	csp_main.i_csp_data_ref^.Production.GoodCasesNoReset	:=	UDINT_TO_DINT(csp_case_main_statistics.logsect.hmi_unresettable_sampled_counters.total_good_products);
	
	csp_main.i_csp_data_ref^.Production.GoodUnitsNoReset	:=	UDINT_TO_DINT(csp_case_main_statistics.logsect.hmi_unresettable_sampled_counters.total_good_products)
																*
																csp_main_brand.case_pattern.case_pattern_L
																*
																csp_main_brand.case_pattern.case_pattern_W;
																
	csp_main.i_csp_data_ref^.Production.TotalUnits			:=	(csp_customerInterfaces.CasePacker.Production.GoodUnits + csp_customerInterfaces.CasePacker.Production.TotalScrapUnits); //Cartoni Ricevuti a monte del metering belt per un ordine, a prescindere che andranno scartati o meno dal pusher
	
	csp_main.i_csp_data_ref^.Production.TotalUnitsNoReset	:=	(
																UDINT_TO_DINT(csp_case_main_statistics.logsect.hmi_unresettable_sampled_counters.total_good_products)
																+
																UDINT_TO_DINT(csp_case_main_statistics.logsect.hmi_unresettable_sampled_counters.total_rejected)
																)
																	*
																	csp_main_brand.case_pattern.case_pattern_L
																	*
																	csp_main_brand.case_pattern.case_pattern_W; //Cartoni Ricevuti a monte del metering belt, a prescindere che andranno scartati o meno dal pusher
																
	csp_main.i_csp_data_ref^.Production.TotalScrapUnits		:=	UDINT_TO_DINT(csp_case_main_statistics.logsect.hmi_shift_independent_sampled_counters.total_rejected)
																*
																csp_main_brand.case_pattern.case_pattern_L
																*
																csp_main_brand.case_pattern.case_pattern_W;
																
	csp_main.i_csp_data_ref^.Production.TotalOrderTime		:= 	UDINT_TO_DINT(mes_elapsed_time_1_npr / 60); 	
	csp_main.i_csp_data_ref^.Production.TotalRunningTime 	:=	UDINT_TO_DINT(mes_elapsed_time_2_npr / 60); 
	
	//Divide by zero protections
	IF UDINT_TO_DINT(csp_case_main_statistics.logsect.hmi_shift_independent_sampled_counters.total_good_products) <> 0
	THEN
	csp_main.i_csp_data_ref^.Production.PercentScrapUnits	:=	(		//Rejected Cases
																		UDINT_TO_DINT(csp_case_main_statistics.logsect.hmi_shift_independent_sampled_counters.total_rejected)
																		/ 
																		UDINT_TO_DINT(csp_case_main_statistics.logsect.hmi_shift_independent_sampled_counters.total_good_products)
																)		//Good Cases
																*
																100;
	END_IF																
	
	csp_main.i_csp_data_ref^.Production.Rejects.Infeed_waterfall	:=	//Barcode Rejects
																		UDINT_TO_DINT(csp_case_main_statistics.logsect.hmi_shift_independent_sampled_counters.auxiliary_counters[1])
																		+
																		//High Load Rejects
																		UDINT_TO_DINT(csp_case_main_statistics.logsect.hmi_shift_independent_sampled_counters.auxiliary_counters[2]);
																			
	csp_main.i_csp_data_ref^.Production.Rejects.Accumulator	:=		//Crosspush Low-load
																		UDINT_TO_DINT(csp_case_main_statistics.logsect.hmi_shift_independent_sampled_counters.auxiliary_counters[3])
																		+
																	//Crosspush High-load
																		UDINT_TO_DINT(csp_case_main_statistics.logsect.hmi_shift_independent_sampled_counters.auxiliary_counters[4]);												
																			
	csp_main.i_csp_data_ref^.Production.Rejects.Case_Feed	:=		//Case Feed Reject
																		UDINT_TO_DINT(csp_case_main_statistics.logsect.hmi_shift_independent_sampled_counters.auxiliary_counters[5]);

	csp_main.i_csp_data_ref^.Production.Rejects.Discharge	:=		//Rejected cases at discharge
																		UDINT_TO_DINT(csp_case_main_statistics.logsect.hmi_shift_independent_sampled_counters.total_rejected);
	
	csp_main.i_csp_data_ref^.Production.Rejects.TBD5		:=		TEST_DINT;
	csp_main.i_csp_data_ref^.Production.Rejects.Sample		:=		TEST_DINT;
	
	(*from RAJones MIX - MARCO *)
	
	csp_main.i_csp_data_ref^.Start.PeakWait 				:= 	FALSE;
	csp_main.i_csp_data_ref^.Start.Ramp 					:= 	FALSE;	
	csp_main.i_csp_data_ref^.Start.Request 					:= 	FALSE;	
	
	csp_main.i_csp_data_ref^.Status.NextJob 				:= 	TEST_DINT;;
	csp_main.i_csp_data_ref^.Status.Running 				:= 	motorization_manager_is_execute(csp_main_motorization_manager.motm);

	csp_main.i_csp_data_ref^.Status.Blocked.Downstream 		:= 	message_is_on(csp_case_discharge_reject_sensors.downstream_backup_hold_aem);
	csp_main.i_csp_data_ref^.Status.Blocked.Reject 			:= 	message_is_on(csp_case_discharge_reject_sensors.consecutive_blocked_reject_aem);
	csp_main.i_csp_data_ref^.Status.Blocked.Waste 			:= 	message_is_on(csp_transfer_crosspusher_reject.backup_di_dchk.alarm_asm.message)
																OR
																message_is_on(csp_transfer_infeed_reject.bin_full_dchk.alarm_asm.message);

	csp_main.i_csp_data_ref^.Status.Faulted.CaseBlanks		:= 	csp_case_feed_magazine.AML_Faulted;;
	
	csp_main.i_csp_data_ref^.Status.Faulted.Main 			:= 	machine_is_stopped(csp.mch)
																AND 
																csp_main_interface.alarm_id <> 430 // SERVICE CYCLE STOP FOR CASE SIDE
																AND 
																csp_main_interface.alarm_id <> 431 // CYCLE STOP FOR CASE SIDE	
																AND 
																csp_main_interface.alarm_id <> 768 // SERVICE CYCLE STOP FOR TRANSFER SIDE
																AND 
																csp_main_interface.alarm_id <> 769;// CYCLE STOP FOR TRANSFER SIDE	

	csp_main.i_csp_data_ref^.Status.Rate.Actual				:= 	LREAL_TO_INT(csp_main_motorization_manager.motm.actual_velocity);
	
	csp_main.i_csp_data_ref^.Status.Rate.Target				:= 	LREAL_TO_INT(csp_main_motorization_manager.motm.actual_velocity_setpoint);
	
	csp_main.i_csp_data_ref^.Status.Starved.CaseBlanks 		:= 	message_is_on(csp_case_feed_magazine_level_zonemin.magazine_level_zone_min_wem); //MARCO: PE presente nella presa cases
	csp_main.i_csp_data_ref^.Status.Starved.Glue 			:= 	NOT digital_input_is_active(csp_case_glue_hotmelt.level_ok_di);
	csp_main.i_csp_data_ref^.Status.Starved.Labels 			:= 	TEST_BOOL; //MARCO: inserire out_of_label che possiamo leggere dallo step 4 della cartoner
	csp_main.i_csp_data_ref^.Status.Starved.Units 			:= 	csp_transfer_infeed_clamp.min_prime; //MARCO: indica che il livello dei cartoni è inferiore al min, oltre ad altri check da verificare se siano corretti (RAJones)
	
	csp_main.i_csp_data_ref^.Status.Stop.AutoReason 		:= 	csp_main_interface.alarm_id; 
	csp_main.i_csp_data_ref^.Status.Stop.Estop 				:= 	//machine_is_stop_emergency_active(csp.mch);
																NOT safety_integrated_series_is_safely_closed(csp_case_main_safety_emergency.sis)
																OR
																NOT safety_integrated_series_is_safely_closed(csp_transfer_main_safety_emergency.sis);
																
	csp_main.i_csp_data_ref^.Status.Stop.Guard 				:= 	NOT safety_integrated_series_is_safely_closed(csp_case_main_safety_guards.sis) OR NOT safety_integrated_series_is_safely_closed(csp_transfer_main_safety_guards.sis);
	csp_main.i_csp_data_ref^.Status.Stop.Operator 			:= 	message_is_on(csp_case_main_services_pushbuttons.stop_dchk.alarm_asm.message)
																OR
																message_is_on(csp_case_main_services_pushbuttons.service_stop_dchk.alarm_asm.message)
																OR
																message_is_on(csp_transfer_main_services_pushbuttons.stop_dchk.alarm_asm.message)
																OR
																message_is_on(csp_transfer_main_services_pushbuttons.service_stop_dchk.alarm_asm.message);
	
	csp_main.i_csp_data_ref^.Status.RunOut 					:= 	csp_main_motorization.empty_command;
	csp_main.i_csp_data_ref^.Status.RunOutComplete 			:=	message_is_on(csp_case_virtualMaster.runout_complete)
																AND csp_case_main_services.end_production
																OR
																p_last_case;
	
ELSE
	mes_elapsed_time_1_npr	:= 0;
	mes_elapsed_time_2_npr	:= 0;
END_IF
END_ACTION

END_PROGRAM

// ---- Application/CSP/Main/Phase Manager/csp_main_phaseManager_run_out.TcPOU
(*********************************** G.D S.p.A. - Technical Department ***********************************
============= PROGRAM INFO ============
FOLDER:             TBD
MACHINES INVOLVED:  TBD 

============= DESCRIPTION =============
WN phase manager program

============= REVISIONS ===============
Date		Version	 	Author      	Description             
----------	-------		------------  	--------------------------------------------
2021/03/18 	0000.01	 	S.Uccellari 	Creation of the PRG
**********************************************************************************************************)
(*$R
	process_ref := prc;
$*)
PROGRAM csp_main_phaseManager_run_out
VAR
	prc:												process;
	prc_path:											STRING;
	
	fsm_enable_conditions:								BOOL;
	fsm_status:											INT;
	
	rejects_for_low_weight_init_cnt:					UDINT;
	rejects_for_low_weight_cnt:							UDINT;	
	rejects_for_low_weight_limit_npr:					UDINT;		(*$P desc := run out - cups under weight; $*)

	confirm_run_out_mode_dpr:							BOOL;		(*$P $*)	
	confirm_run_out_mode_pow:							parameter_overwrite;	
	confirm_run_out_mode_visibility:					INT := 1; 	(*$H_R	desc := visibility; $*)

	low_weight_limit_asm:								message;	
	run_out_complete_asm:								message;	
	
	
	run_out_running:									BOOL;
	run_out_done:										BOOL;
	
END_VAR

_read_var_input();

_object_manager();

IF NOT objects_running()
THEN
	RETURN;	
END_IF

_read_process_image();

_mode_manager();

CASE process_get_mode(prc) of
	MODE_ABSENT,
	MODE_INACTIVE:
		RETURN;
	MODE_TEST:
		_handle_process_test();
END_CASE

_set_runtime_properties();

(********************************* BODY *********************************)

(************************************************************************)

(**************************** PROGRAM HANDLER ***************************)
run_cycle();
(************************************************************************)

_handle_messages();

_write_output();

ACTION _handle_messages:
;
END_ACTION

ACTION _handle_process_test:
;
END_ACTION

ACTION _mode_manager:
IF process_mode_req_is_pending(prc)
THEN
    process_apply_mode_req_first_step(prc);
    CASE process_get_mode(prc) OF
        MODE_TO_ABSENT:
			;
        MODE_TO_INACTIVE:
			;
        MODE_TO_TEST:
			;
        MODE_TO_OPERATIONAL:
			;
    END_CASE
    process_apply_mode_req_second_step(prc);
END_IF
END_ACTION

ACTION _object_manager:
IF objects_initialization()
THEN
	sub_process_init(
		object_name					:= 'csp_main_phaseManager_run_out.prc', 
		process						:= csp_main_phaseManager.prc, 
		CONVERSION_this				:= prc);
		
	prc_path 						:= process_get_path(prc);
	
	parameter_overwrite_bool_init(
		object_name								:= CONCAT(prc_path, '_confirm_run_out_mode_pow'), 
		parameter								:= confirm_run_out_mode_dpr, 
		process									:= prc, 
		CONVERSION_this							:= confirm_run_out_mode_pow);		

	process_message_init(
		object_name					:= CONCAT(prc_path, '_low_weight_limit_asm'), 
		behaviour					:= MESSAGE_BEHAVIOUR_STATE, 
		reset_timeout				:= 0, 
		disableable					:= FALSE, 
		individual_reset			:= FALSE, 
		machine_reaction			:= MACHINE_REACTION_NORMAL_STOP, 
		typology					:= MESSAGE_TYPOLOGY_ABNORMAL, 
		process						:= prc, 
		CONVERSION_this				:= low_weight_limit_asm);

	process_message_init(
		object_name					:= CONCAT(prc_path, '_run_out_complete_asm'), 
		behaviour					:= MESSAGE_BEHAVIOUR_EVENT, 
		reset_timeout				:= 0, 
		disableable					:= FALSE, 
		individual_reset			:= FALSE, 
		machine_reaction			:= MACHINE_REACTION_NORMAL_STOP, 
		typology					:= MESSAGE_TYPOLOGY_ABNORMAL, 
		process						:= prc, 
		CONVERSION_this				:= run_out_complete_asm);


		

END_IF

IF objects_running()
THEN
	process_cycle(prc);
END_IF
END_ACTION

ACTION _read_process_image:
;
END_ACTION

ACTION _read_var_input:
;
END_ACTION

ACTION _set_runtime_properties:
;
END_ACTION

ACTION _write_output:
;
END_ACTION

ACTION run_cycle:
IF	csp_main_phaseManager.fsm_status = CSP_MAIN_PHASE_MANAGER_STATUS_UNDEFINED_0
	AND
	csp_main_phaseManager.p_mes_interface_enable
THEN	
	fsm_status := 0;
END_IF

fsm_enable_conditions :=
	(
		csp_main_phaseManager.fsm_status
		=
		CSP_MAIN_PHASE_MANAGER_STATUS_RUNOUT_60
	);
	
IF	NOT fsm_enable_conditions
THEN
	process_message_reset(low_weight_limit_asm);	
	IF	run_out_running	
	THEN
		fsm_status := 666;
	END_IF;	
END_IF

CASE fsm_status OF
	0:
		confirm_run_out_mode_visibility := 1;	
		csp_main.i_csp_data_ref^.Status.RunOutComplete := FALSE;
		IF fsm_enable_conditions
		THEN
			run_out_done := FALSE;
			run_out_running := TRUE;
			fsm_status := 20;
		END_IF
		
	20:		
		fsm_status := 30;			
		

	30:	
		fsm_status := 40;	

	40:
		confirm_run_out_mode_visibility := 1;
		csp_main.i_csp_data_ref^.Status.RunOut := TRUE; (* use this to empty the filler *)

			fsm_status := 555;


	50: 
		;
		(*IF filler_empty
		THEN
			process_message_set(
				errorID_1			:= 1, 
				errorID_2			:= 0, 
				errorID_3			:= 0, 
				CONVERSION_this		:= run_out_complete_asm);

			run_out step1 AND run out cartoner
			
			fsm_status := 555;
		END_IF*)
		
		
	555:
		csp_main.i_csp_data_ref^.Status.RunOut := FALSE;	
		csp_main.i_csp_data_ref^.Status.RunOutComplete := TRUE;
		run_out_running := FALSE;
		run_out_done := TRUE;
		confirm_run_out_mode_visibility := 1;
		
		IF	csp_main.i_filler_upstream_coffee //MARCO 0904
		THEN
			run_out_running := FALSE;
			run_out_done := FALSE;
			fsm_status := 0;
		END_IF		
		
	666:
		run_out_running := FALSE;
		run_out_done := FALSE;
		confirm_run_out_mode_visibility := 1;		
		csp_main.i_csp_data_ref^.Status.RunOut := FALSE;		
		csp_main.i_csp_data_ref^.Status.RunOutComplete := FALSE;
		//IF NOT csp_main.i_upstream_coffee^.Down //MARCO 0904
		//THEN
			fsm_status := 0;
		//END_IF
END_CASE
END_ACTION

END_PROGRAM

// ---- Application/CSP/Main/Phase Manager/Snapshot/csp_main_phaseManager_set_snapshot.TcPOU
(*********************************** G.D S.p.A. - Technical Department ***********************************
============= PROGRAM INFO ============
FOLDER:             TBD
MACHINES INVOLVED:  TBD 

============= DESCRIPTION =============
WU phase manager snapshot set function

============= REVISIONS ===============
Date		Version	 	Author      	Description             
----------	-------		------------  	--------------------------------------------
2020/06/19 	0000.00	 	G.Cera 			Creation of the PRG

**********************************************************************************************************)

FUNCTION csp_main_phaseManager_set_snapshot : VOID
VAR_INPUT
    errorID_1:				DINT;			(* Field for specify the faults code or enter
								   				more message info *)
    errorID_2:				DINT;			(* Field for specify the faults code or enter
								   				more message info *)
    errorID_3:				DINT;			(* Field for specify the faults code or enter
								   				more message info *)
	reason:					STRING := '';

	job_not_scheduled:		BOOL;
	
	job_pending:			BOOL;
	
END_VAR

VAR_IN_OUT
    CONVERSION_this:		csp_main_phaseManager_snapshot;
								(* csp_main_phaseManager_snapshot snapshot reference *)
END_VAR

IF	message_set(
		errorID_1		:= errorID_1, 
		errorID_2		:= errorID_2, 
		errorID_3		:= errorID_3, 
		CONVERSION_this	:= CONVERSION_this.message)
THEN
	CONVERSION_this.reason 				:= reason;
	CONVERSION_this.job_not_scheduled	:= job_not_scheduled;
	CONVERSION_this.job_pending			:= job_pending;
END_IF

END_FUNCTION

// ---- Application/CSP/Main/Phase Manager/Snapshot/csp_main_phaseManager_warning_set_snapshot.TcPOU
(*********************************** G.D S.p.A. - Technical Department ***********************************
============= PROGRAM INFO ============
FOLDER:             TBD
MACHINES INVOLVED:  TBD 

============= DESCRIPTION =============
WU phase manager snapshot set function

============= REVISIONS ===============
Date		Version	 	Author      	Description             
----------	-------		------------  	--------------------------------------------
2020/06/19 	0000.00	 	G.Cera 			Creation of the PRG

**********************************************************************************************************)

FUNCTION csp_main_phaseManager_warning_set_snapshot : VOID
VAR_INPUT
    errorID_1:				DINT;			(* Field for specify the faults code or enter
								   				more message info *)
    errorID_2:				DINT;			(* Field for specify the faults code or enter
								   				more message info *)
    errorID_3:				DINT;			(* Field for specify the faults code or enter
								   				more message info *)
	reason:					STRING := '';

	maintenance_job_active:	BOOL;
		
END_VAR

VAR_IN_OUT
    CONVERSION_this:		csp_main_phaseManager_warning_snapshot;
								(* csp_main_phaseManager_snapshot snapshot reference *)
END_VAR

IF	message_set(
		errorID_1		:= errorID_1, 
		errorID_2		:= errorID_2, 
		errorID_3		:= errorID_3, 
		CONVERSION_this	:= CONVERSION_this.message)
THEN
	CONVERSION_this.w_reason 					:= reason;
	CONVERSION_this.maintenance_job_active	:= maintenance_job_active;
END_IF

END_FUNCTION

// ---- Application/CSP/Main/Phase Manager/Snapshot/csp_main_phMan_start_job_set_snapshot.TcPOU
(*********************************** G.D S.p.A. - Technical Department ***********************************
============= PROGRAM INFO ============
FOLDER:             TBD
MACHINES INVOLVED:  TBD 

============= DESCRIPTION =============
WU phase manager snapshot set function

============= REVISIONS ===============
Date		Version	 	Author      	Description             
----------	-------		------------  	--------------------------------------------
2020/06/19 	0000.00	 	G.Cera 			Creation of the PRG

**********************************************************************************************************)

FUNCTION csp_main_phMan_start_job_set_snapshot : VOID
VAR_INPUT
    errorID_1:				DINT;			(* Field for specify the faults code or enter
								   				more message info *)
    errorID_2:				DINT;			(* Field for specify the faults code or enter
								   				more message info *)
    errorID_3:				DINT;			(* Field for specify the faults code or enter
								   				more message info *)
	reason:					STRING := '';

	order_valid:			BOOL;
	
	product_valid:			BOOL;
	
	recipe_valid:			BOOL;
	
	materials_valid:		BOOL;
	
	mark_valid:				BOOL;	
	
END_VAR

VAR_IN_OUT
    CONVERSION_this:		csp_main_phMan_start_job_snapshot;
								(* csp_main_phaseManager_snapshot snapshot reference *)
END_VAR

IF	message_set(
		errorID_1		:= errorID_1, 
		errorID_2		:= errorID_2, 
		errorID_3		:= errorID_3, 
		CONVERSION_this	:= CONVERSION_this.message)
THEN
	CONVERSION_this.sj_reason 				:= reason;
	CONVERSION_this.order_valid			:= order_valid;
	CONVERSION_this.recipe_valid		:= recipe_valid;
	CONVERSION_this.product_valid		:= product_valid;
	CONVERSION_this.materials_valid		:= materials_valid;
	CONVERSION_this.mark_valid			:= mark_valid;
END_IF

END_FUNCTION

// ---- Application/CSP/Main/Phase Manager/Snapshot/csp_main_phMan_start_job_init_snapshot.TcPOU
(*********************************** G.D S.p.A. - Technical Department ***********************************
============= PROGRAM INFO ============
FOLDER:             TBD
MACHINES INVOLVED:  TBD 

============= DESCRIPTION =============
WU phase manager snapshot init function

============= REVISIONS ===============
Date		Version	 	Author      	Description             
----------	-------		------------  	--------------------------------------------
2020/06/19 	0000.00	 	G.Cera 			Creation of the PRG

**********************************************************************************************************)

FUNCTION csp_main_phMan_start_job_init_snapshot : VOID
VAR_INPUT	
	message_name:			STRING(MAX_OBJ_NAME_LENGTH);
	behaviour:				message_behaviour_enum;			(* Message type. State or event *)
	reset_timeout:			UDINT;							(* Timeout of reset attempt valid for messages
															   with <a href="#message_behaviour_enum"><i>behaviour</i></a>
															   = MESSAGE_BEHAVIOUR_TRY_AND_CHECK *)
    disableable:        	BOOL;							(* Indicates the possibility
																to disable the message by HMI *)
    individual_reset:   	BOOL;							(* Need explicit reset by
																HMI for acknowlege the message.
																TRUE = individual_reset *)
    machine_reaction:		machine_reaction_enum;			(* Machine stop type.(emergency, normal,
																on phase, ...) *)
    typology:				message_typology_enum;			(* <a href="#message_typology_enum"><i>typology</i></a> *)	
END_VAR

VAR_IN_OUT
    process:                process;                    	(*$ <a href="#process_object"><i>process</i></a> membership $*)
	CONVERSION_this:		csp_main_phMan_start_job_snapshot;			
END_VAR

process_message_init(
	object_name 		:= message_name,
	behaviour 			:= behaviour,
	reset_timeout 		:= reset_timeout,
	disableable 		:= disableable,
	individual_reset 	:= individual_reset,
	machine_reaction 	:= machine_reaction,
	typology			:= typology,
	process 			:= process,
	CONVERSION_this 	:= CONVERSION_this.message);

CONVERSION_this.sj_reason := '';
CONVERSION_this.order_valid := FALSE;
CONVERSION_this.product_valid := FALSE;
CONVERSION_this.recipe_valid := FALSE;
CONVERSION_this.materials_valid := FALSE;
CONVERSION_this.mark_valid := FALSE;

END_FUNCTION

// ---- Application/CSP/Main/Phase Manager/Snapshot/csp_main_phaseManager_init_snapshot.TcPOU
(*********************************** G.D S.p.A. - Technical Department ***********************************
============= PROGRAM INFO ============
FOLDER:             TBD
MACHINES INVOLVED:  TBD 

============= DESCRIPTION =============
WU phase manager snapshot init function

============= REVISIONS ===============
Date		Version	 	Author      	Description             
----------	-------		------------  	--------------------------------------------
2020/06/19 	0000.00	 	G.Cera 			Creation of the PRG

**********************************************************************************************************)

FUNCTION csp_main_phaseManager_init_snapshot : VOID
VAR_INPUT	
	message_name:			STRING(MAX_OBJ_NAME_LENGTH);
	behaviour:				message_behaviour_enum;			(* Message type. State or event *)
	reset_timeout:			UDINT;							(* Timeout of reset attempt valid for messages
															   with <a href="#message_behaviour_enum"><i>behaviour</i></a>
															   = MESSAGE_BEHAVIOUR_TRY_AND_CHECK *)
    disableable:        	BOOL;							(* Indicates the possibility
																to disable the message by HMI *)
    individual_reset:   	BOOL;							(* Need explicit reset by
																HMI for acknowlege the message.
																TRUE = individual_reset *)
    machine_reaction:		machine_reaction_enum;			(* Machine stop type.(emergency, normal,
																on phase, ...) *)
    typology:				message_typology_enum;			(* <a href="#message_typology_enum"><i>typology</i></a> *)	
END_VAR

VAR_IN_OUT
    process:                process;                    	(*$ <a href="#process_object"><i>process</i></a> membership $*)
	CONVERSION_this:		csp_main_phaseManager_snapshot;			
END_VAR

process_message_init(
	object_name 		:= message_name,
	behaviour 			:= behaviour,
	reset_timeout 		:= reset_timeout,
	disableable 		:= disableable,
	individual_reset 	:= individual_reset,
	machine_reaction 	:= machine_reaction,
	typology			:= typology,
	process 			:= process,
	CONVERSION_this 	:= CONVERSION_this.message);

CONVERSION_this.reason := '';
CONVERSION_this.job_not_scheduled := FALSE;
CONVERSION_this.job_pending := FALSE;

END_FUNCTION

// ---- Application/CSP/Main/Phase Manager/Snapshot/csp_main_phaseManager_warning_init_snapshot.TcPOU
(*********************************** G.D S.p.A. - Technical Department ***********************************
============= PROGRAM INFO ============
FOLDER:             TBD
MACHINES INVOLVED:  TBD 

============= DESCRIPTION =============
WU phase manager snapshot init function

============= REVISIONS ===============
Date		Version	 	Author      	Description             
----------	-------		------------  	--------------------------------------------
2020/06/19 	0000.00	 	G.Cera 			Creation of the PRG

**********************************************************************************************************)

FUNCTION csp_main_phaseManager_warning_init_snapshot : VOID
VAR_INPUT	
	message_name:			STRING(MAX_OBJ_NAME_LENGTH);
	behaviour:				message_behaviour_enum;			(* Message type. State or event *)
	reset_timeout:			UDINT;							(* Timeout of reset attempt valid for messages
															   with <a href="#message_behaviour_enum"><i>behaviour</i></a>
															   = MESSAGE_BEHAVIOUR_TRY_AND_CHECK *)
    disableable:        	BOOL;							(* Indicates the possibility
																to disable the message by HMI *)
    individual_reset:   	BOOL;							(* Need explicit reset by
																HMI for acknowlege the message.
																TRUE = individual_reset *)
    machine_reaction:		machine_reaction_enum;			(* Machine stop type.(emergency, normal,
																on phase, ...) *)
    typology:				message_typology_enum;			(* <a href="#message_typology_enum"><i>typology</i></a> *)	
END_VAR

VAR_IN_OUT
    process:                process;                    	(*$ <a href="#process_object"><i>process</i></a> membership $*)
	CONVERSION_this:		csp_main_phaseManager_warning_snapshot;			
END_VAR

process_message_init(
	object_name 		:= message_name,
	behaviour 			:= behaviour,
	reset_timeout 		:= reset_timeout,
	disableable 		:= disableable,
	individual_reset 	:= individual_reset,
	machine_reaction 	:= machine_reaction,
	typology			:= typology,
	process 			:= process,
	CONVERSION_this 	:= CONVERSION_this.message);

CONVERSION_this.w_reason := '';
CONVERSION_this.maintenance_job_active := FALSE;

END_FUNCTION

// ---- Application/CSP/Main/Phase Manager/csp_main_phaseManager_end_job.TcPOU
(*********************************** G.D S.p.A. - Technical Department ***********************************
============= PROGRAM INFO ============
FOLDER:             TBD
MACHINES INVOLVED:  TBD 

============= DESCRIPTION =============
WN phase manager program

============= REVISIONS ===============
Date		Version	 	Author      	Description             
----------	-------		------------  	--------------------------------------------
2021/03/18 	0000.01	 	S.Uccellari 	Creation of the PRG
**********************************************************************************************************)
(*$R
	process_ref := prc;
$*)
PROGRAM csp_main_phaseManager_end_job
VAR
	prc:												process;
	prc_path:											STRING;
	
	fsm_enable_conditions:								BOOL;
	fsm_status:											INT;
	
	cycle_disable_from_mes_asm:							message;	
	
	end_job_running:									BOOL;
	end_job_done:										BOOL;
	
	i_start_job_done:									POINTER TO BOOL;	
	i_run_out_done:										POINTER TO BOOL;	
	
	debug_mes_endJobReq:								BOOL;		
	
END_VAR

_read_var_input();

_object_manager();

IF NOT objects_running()
THEN
	RETURN;	
END_IF

_read_process_image();

_mode_manager();

CASE process_get_mode(prc) of
	MODE_ABSENT,
	MODE_INACTIVE:
		RETURN;
	MODE_TEST:
		_handle_process_test();
END_CASE

_set_runtime_properties();

(********************************* BODY *********************************)

(************************************************************************)

(**************************** PROGRAM HANDLER ***************************)
run_cycle();
(************************************************************************)

_handle_messages();

_write_output();

ACTION _handle_messages:
;
END_ACTION

ACTION _handle_process_test:
;
END_ACTION

ACTION _mode_manager:
IF process_mode_req_is_pending(prc)
THEN
    process_apply_mode_req_first_step(prc);
    CASE process_get_mode(prc) OF
        MODE_TO_ABSENT:
			;
        MODE_TO_INACTIVE:
			;
        MODE_TO_TEST:
			;
        MODE_TO_OPERATIONAL:
			;
    END_CASE
    process_apply_mode_req_second_step(prc);
END_IF
END_ACTION

ACTION _object_manager:
IF objects_initialization()
THEN
	sub_process_init(
		object_name					:= 'csp_main_phaseManager_end_job.prc', 
		process						:= csp_main_phaseManager.prc, 
		CONVERSION_this				:= prc);
		
	prc_path 						:= process_get_path(prc);
	
	process_message_init(
		object_name					:= CONCAT(prc_path, '_cycle_disable_from_mes_asm'), 
		behaviour					:= MESSAGE_BEHAVIOUR_EVENT, 
		reset_timeout				:= 0, 
		disableable					:= FALSE, 
		individual_reset			:= FALSE, 
		machine_reaction			:= MACHINE_REACTION_NORMAL_STOP, 
		typology					:= MESSAGE_TYPOLOGY_ABNORMAL, 
		process						:= prc, 
		CONVERSION_this				:= cycle_disable_from_mes_asm);



END_IF

IF objects_running()
THEN
	process_cycle(prc);
END_IF
END_ACTION

ACTION _read_process_image:
;
END_ACTION

ACTION _read_var_input:
i_start_job_done 	:= ADR(csp_main_phaseManager_startJob.start_job_done);
i_run_out_done		:= ADR(csp_main_phaseManager_run_out.run_out_done);
END_ACTION

ACTION _set_runtime_properties:
;
END_ACTION

ACTION _write_output:
;
END_ACTION

ACTION run_cycle:
IF	csp_main_phaseManager.fsm_status = CSP_MAIN_PHASE_MANAGER_STATUS_UNDEFINED_0
THEN	
	fsm_status := 0;
END_IF

fsm_enable_conditions :=
	(
		csp_main_phaseManager.fsm_status
		=
		CSP_MAIN_PHASE_MANAGER_STATUS_END_JOB_70
	);
	
IF	NOT fsm_enable_conditions
THEN
	IF	end_job_running	
	THEN
		fsm_status := 666;
	END_IF;	
END_IF

CASE fsm_status OF
	0:	
		IF	fsm_enable_conditions
		THEN
				process_message_set(
					errorID_1			:= 1, 
					errorID_2			:= 0, 
				errorID_3			:= 0, 
					CONVERSION_this		:= cycle_disable_from_mes_asm);		
			
				end_job_done := FALSE;
				end_job_running := TRUE;
				fsm_status := 10;	
		END_IF	
		
	
	10:
		IF	csp_main.i_end_job_request
		THEN	
			log_section_upd_and_reset_factory_driven(csp_case_main_statistics.logsect);				
			csp_main.i_csp_data_ref^.Status.Job := 1;
			csp_main.i_cartons_count := 0;
			csp_main.i_cartoner_RunOutComplete:= FALSE;
			csp_main.i_csp_data_ref^.Status.RunOutComplete := FALSE;
			//Reset MES variables
			
			csp_main.i_mark_bubd_information^.BestUsedByDate 	:= '';
			csp_main.i_mark_bubd_information^.Prefix 			:= '';
			csp_main.i_mark_information^.ID 					:= '';
			csp_main.i_mark_information^.KdpSite 				:= '';
			csp_main.i_mark_information^.OriginDate 			:= '';
			csp_main.i_mark_information^.PartnerSite			:= '';
			csp_main.i_mark_information^.Template.Carton		:= '';
			csp_main.i_mark_information^.Template.CASEPACK		:= '';
			csp_main.i_mark_information^.Template.Pod			:= '';			
			
			csp_main.i_current_material_information^[csp_main_phaseManager.MASTER_CASE_BLANK_MATERIAL_ID].ID 	:= '';
			csp_main.i_current_material_information^[csp_main_phaseManager.MASTER_CASE_BLANK_MATERIAL_ID].QTY	:= 0;
			csp_main.i_next_material_information^[csp_main_phaseManager.MASTER_CASE_BLANK_MATERIAL_ID].ID		:= '';
			csp_main.i_next_material_information^[csp_main_phaseManager.MASTER_CASE_BLANK_MATERIAL_ID].QTY		:= 0;
            
			csp_main.i_current_material_information^[csp_main_phaseManager.CASE_LABEL_MATERIAL_ID].ID 			:= '';
			csp_main.i_current_material_information^[csp_main_phaseManager.CASE_LABEL_MATERIAL_ID].QTY			:= 0;
			csp_main.i_next_material_information^[csp_main_phaseManager.CASE_LABEL_MATERIAL_ID].ID				:= '';
			csp_main.i_next_material_information^[csp_main_phaseManager.CASE_LABEL_MATERIAL_ID].QTY				:= 0;

			csp_main.i_next_recipe_information^.CasePacker														:= '';
			csp_main.i_recipe_information^.CasePacker															:= '';			
			csp_main.i_next_recipe_information^.Filler															:= '';
			csp_main.i_recipe_information^.Filler																:= '';
			csp_main.i_next_recipe_information^.Cartoner														:= '';
			csp_main.i_recipe_information^.Cartoner																:= '';			

			csp_main.i_order_information^.ID																	:= '';	
			csp_main.i_order_information^.SapBatchID															:= '';			
			csp_main.i_next_order_information^.ID						:= '';	
			csp_main.i_next_order_information^.SapBatchID				:= '';			
			
			csp_main.i_csp_data_ref^.Production.GoodCases				:= 0;
			
			csp_main.i_product_information^.CaffeinatedFlag				:= FALSE;
			csp_main.i_product_information^.CartonsPerCase				:= 0;
			csp_main.i_product_information^.FillWeight.Maximum			:= 0;
			csp_main.i_product_information^.FillWeight.Minimum			:= 0;
			csp_main.i_product_information^.FillWeight.Target			:= 0;
			csp_main.i_product_information^.FilterType					:= '';
			csp_main.i_product_information^.FlavorDose					:= 0;
			csp_main.i_product_information^.FlavorFlag					:= FALSE;
			csp_main.i_product_information^.ID							:= '';
			csp_main.i_product_information^.UPC							:= '';
			csp_main.i_product_information^.KosherFlag					:= FALSE;
			csp_main.i_product_information^.OrganicFlag					:= FALSE;
			csp_main.i_product_information^.PodsPerCarton				:= 0;
			csp_main.i_product_information^.PodsPerCase					:= 0;
			csp_main.i_product_information^.ShelfLife					:= 0;			
			csp_main.i_next_product_information^.CaffeinatedFlag		:= FALSE;
			csp_main.i_next_product_information^.CartonsPerCase			:= 0;
			csp_main.i_next_product_information^.FillWeight.Maximum		:= 0;
			csp_main.i_next_product_information^.FillWeight.Minimum		:= 0;
			csp_main.i_next_product_information^.FillWeight.Target		:= 0;
			csp_main.i_next_product_information^.FilterType				:= '';
			csp_main.i_next_product_information^.FlavorDose				:= 0;
			csp_main.i_next_product_information^.FlavorFlag				:= FALSE;
			csp_main.i_next_product_information^.ID						:= '';
			csp_main.i_next_product_information^.UPC					:= '';
			csp_main.i_next_product_information^.KosherFlag				:= FALSE;
			csp_main.i_next_product_information^.OrganicFlag			:= FALSE;
			csp_main.i_next_product_information^.PodsPerCarton			:= 0;
			csp_main.i_next_product_information^.PodsPerCase			:= 0;
			csp_main.i_next_product_information^.ShelfLife				:= 0;					
			csp_main.i_csp_data_ref^.CaseBlanks.ConsumedCart			:= 0;			
			csp_main.i_csp_data_ref^.CaseBlanks.ConsumedTotal			:= 0;
			csp_main.i_csp_data_ref^.Labels.Consumed					:= 0;
			
			parameter_overwrite_set_bool_value(
					value				:= FALSE, 
					CONVERSION_this		:= csp_main_phaseManager.confirm_run_out_mode_pow);			

			//IF csp_case_main_statistics.logsect.customer_driven_update_and_reset_received
			//THEN
			fsm_status := 555;
			//END_IF
						
		END_IF
	
		
	555:
		i_start_job_done^ := FALSE;
		i_run_out_done^ := FALSE;	
		end_job_done := TRUE;
		end_job_running := FALSE;
		
	
		
	666:
		i_start_job_done^ := FALSE;
		i_run_out_done^ := FALSE;		
		end_job_running := FALSE;
		end_job_done := FALSE;
		fsm_status := 0;

END_CASE
END_ACTION

END_PROGRAM

// ---- Application/CSP/Case/Glue/HotMelt/csp_case_glue_hotMelt.TcPOU
(*********************************** G.D S.p.A. - Technical Department ***********************************
============= PROGRAM INFO ============
FOLDER:             TBD
MACHINES INVOLVED:  TBD 

============= DESCRIPTION =============
csp machine declaration

============= REVISIONS ===============
Date		Version	 	Author      	Description             
----------	-------		------------  	--------------------------------------------
2020/02/24 	0001.00	 	G.Imbriaco		Hotmelt System. Ready, Level and Standby req.

**********************************************************************************************************)
(*$R process_ref := prc; $*)
PROGRAM csp_case_glue_hotMelt
VAR
	
	prc:											process;
	prc_path:										STRING;
	
	level_ok_di:									digital_input;
	level_ok_dchk:									digital_check;
	
	level_stop_cur_cycles:							DINT:=0;
	level_stop_max_cycles:							DINT := 25;
	
	level_stop_asm:									message;
	
	ready_di:										digital_input;
	ready_dchk:										digital_check;

	standby_req:									BOOL:=FALSE;(*$P $*)
	standby_command:								BOOL:=FALSE;
	
	standby_do:										digital_output;
	standby_sact:									digital_actuator;
	standby_active_wsm:								message;
	
	glue_standby_ton: 								TON;
	standby_delay_bool:								BOOL;
	standby_delay_ton_complete: 					BOOL := FALSE;
	glue_standby_resend_ton: 						Ton;
	Standby_timeout_elapsed: 						STRING;	(*$P desc := Elapsed Time of glue standby timeout. 1 Hour is limit; $*)
	Standby_status: 								STRING;	(*$P desc := Status of the glue standby reqeuest; $*)

	feeder_faulted_di:								digital_input;
	feeder_faulted_dchk:							digital_check;
	
	Standby_timeout_min:							DINT := 60; (*$P $*)
	Standby_timeout_ms:								DINT;
	glue_standby_ton_PT: 							TIME;

END_VAR

VAR CONSTANT
	LEVEL_ALARM_DELAY_MS:							INT := 1000;
	READY_ALARM_DELAY_MS:							DINT := 500;
	
	ENABLE_SACT_ACTIVATION_TIME_MS:					UDINT := 100;
	ENABLE_SACT_DEACTIVATION_TIME_MS:				UDINT := 100;
END_VAR

_read_var_input();

_object_manager();

IF NOT objects_running()
THEN
	RETURN;	
END_IF

_read_process_image();

_mode_manager();

CASE process_get_mode(prc) of
	MODE_ABSENT,
	MODE_INACTIVE:
		RETURN;
	MODE_TEST:
		_handle_process_test();
END_CASE

_set_runtime_properties();

(********************************* BODY *********************************)

Standby_timeout_ms := Standby_timeout_min * 60000; //Converts Minutes to MS for timer
glue_standby_ton_PT := DINT_TO_TIME(Standby_timeout_ms);

(* standby logic to start the timer for standby command*)
IF csp.o_machine_is_stopped
	AND NOT csp.i_reset_button
THEN
	standby_delay_bool := TRUE;
ELSE
	standby_delay_bool := FALSE;
END_IF

(* standby timer if case packer is stopped for an hour*)
glue_standby_ton(IN:=standby_delay_bool , PT:= glue_standby_ton_PT , Q=> , ET=> );
(* standby timer checks every 10min if case packer is stopped for an hour and no reset command*)
glue_standby_resend_ton(IN:=(standby_req AND NOT glue_standby_resend_ton.Q) , PT:= T#10M , Q=> , ET=> );

Standby_timeout_elapsed := TIME_TO_STRING(glue_standby_ton.ET);
	
(* standby_command := button_is_pressed( XXXX ); In case of hardware button for standby *)
IF standby_command
THEN
	digital_actuator_deactivate(standby_sact);//De-activation puts Hotmelt unit in Standby mode
	(* button_lamp_blink(XXXX);*)
	process_message_set(0, 0, 0, standby_active_wsm);
	Standby_status := 'Standby Active';
ELSE
	digital_actuator_activate(standby_sact); //Activation takes Hotmelt Unit out of Standby mode
	(* button_lamp_on(XXXX); *)
	process_message_reset(standby_active_wsm);
	Standby_status := 'Standby Not Active';
END_IF
	
(* standby set command if timer is completed*)
IF glue_standby_ton.q
	OR
		(standby_req
		AND
		glue_standby_resend_ton.Q)
THEN
		standby_req := TRUE;
END_IF

(* standby reset command if reset is pushed or command on HMI*)
IF csp.i_reset_button
THEN
	standby_req := FALSE;
END_IF

IF digital_check_is_ok(level_ok_dchk)
THEN
	level_stop_cur_cycles := 0;
	process_message_reset(level_stop_asm);
ELSE
	IF phase_edge(csp_case_transport_virtualMaster.transport_vm_ph)
	THEN		
		level_stop_cur_cycles := level_stop_cur_cycles + 1;
		
		IF level_stop_cur_cycles > level_stop_max_cycles
		THEN
			//stop machine due to low glue
			process_message_set(1,0,0,level_stop_asm);
		END_IF
	END_IF
END_IF

(************************************************************************)

_handle_messages();

_write_output();

ACTION _handle_messages:
IF	standby_command
THEN
	process_message_set(
		errorID_1		:= 1, 
		errorID_2		:= 0, 
		errorID_3		:= 0, 
		CONVERSION_this	:= standby_active_wsm);
ELSE
	process_message_reset(standby_active_wsm);
END_IF
END_ACTION

ACTION _handle_process_test:
;
END_ACTION

ACTION _mode_manager:
IF process_mode_req_is_pending(prc)
THEN
    process_apply_mode_req_first_step(prc);
    CASE process_get_mode(prc) OF
        MODE_TO_ABSENT:
			;
        MODE_TO_INACTIVE:
			;
        MODE_TO_TEST:
			;
        MODE_TO_OPERATIONAL:
			;
    END_CASE
    process_apply_mode_req_second_step(prc);
END_IF
END_ACTION

ACTION _object_manager:
IF objects_initialization()
THEN
	sub_process_init(
		object_name						:= 'csp_case_glue_hotMelt.prc', 
		process							:= csp_case_glue.prc, 
		CONVERSION_this					:= prc);
		
	prc_path 							:= process_get_path(prc);
	
	(* HHS HOT MELT TANK INTERFACE *)
	
	digital_input_init(
		object_name						:= CONCAT(prc_path, '_level_ok_di'), 
		polarity_direct					:= TRUE, 
		process							:= prc, 
		CONVERSION_this					:= level_ok_di);
	
	digital_check_and_message_init(
		object_name						:= CONCAT(prc_path, '_level_ok_dchk'), 
		alarm_if_input_off				:= TRUE, 
		alarm_delay						:= LEVEL_ALARM_DELAY_MS, 
		enabled_at_powerup				:= TRUE, 
		individual_reset				:= FALSE, 
		machine_reaction				:= MACHINE_REACTION_NO_STOP, 
		typology						:= MESSAGE_TYPOLOGY_NORMAL, 
		process							:= prc, 
		CONVERSION_this					:= level_ok_dchk);
		
	digital_check_add_di(
		di								:= level_ok_di, 
		CONVERSION_this					:= level_ok_dchk);
		
	digital_input_init(
		object_name						:= CONCAT(prc_path, '_ready_di'), 
		polarity_direct					:= TRUE, 
		process							:= prc, 
		CONVERSION_this					:= ready_di);
	
	digital_check_and_message_init(
		object_name						:= CONCAT(prc_path, '_ready_dchk'), 
		alarm_if_input_off				:= TRUE, 
		alarm_delay						:= READY_ALARM_DELAY_MS, 
		enabled_at_powerup				:= TRUE, 
		individual_reset				:= FALSE, 
		machine_reaction				:= MACHINE_REACTION_STOP_IN_PHASE_ONE, 
		typology						:= MESSAGE_TYPOLOGY_ABNORMAL, 
		process							:= prc, 
		CONVERSION_this					:= ready_dchk);

	digital_check_add_di(
		di								:= ready_di, 
		CONVERSION_this					:= ready_dchk);	
		

	digital_output_init(
		object_name						:= CONCAT(prc_path, '_standby_do'), 
		polarity_direct					:= TRUE, 
		process							:= prc, 
		CONVERSION_this					:= standby_do);

	digital_actuator_init(
		object_name						:= CONCAT(prc_path, '_standby_sact'), 
		_type							:= DIGITAL_ACTUATOR_TYPE_IN_xx, 
		fault_reaction					:= DIGITAL_ACTUATOR_FAULT_REACTION_DEACTIVATING, 
		active_time						:= ENABLE_SACT_ACTIVATION_TIME_MS, 
		inactive_time					:= ENABLE_SACT_DEACTIVATION_TIME_MS, 
		dout							:= standby_do, 
		process							:= prc, 
		CONVERSION_this					:= standby_sact);	

	process_message_init(
		object_name						:= CONCAT(prc_path, '_standby_active_wsm'), 
		behaviour						:= MESSAGE_BEHAVIOUR_STATE, 
		reset_timeout					:= 0, 
		disableable						:= FALSE, 
		individual_reset				:= FALSE, 
		machine_reaction				:= MACHINE_REACTION_STOP_IN_PHASE_ONE, 
		typology						:= MESSAGE_TYPOLOGY_ABNORMAL, 
		process							:= prc, 
		CONVERSION_this					:= standby_active_wsm);
		
	process_message_init(
		object_name						:= CONCAT(prc_path, '_level_stop_asm'), 
		behaviour						:= MESSAGE_BEHAVIOUR_STATE, 
		reset_timeout					:= 0, 
		disableable						:= TRUE, 
		individual_reset				:= FALSE, 
		machine_reaction				:= MACHINE_REACTION_STOP_IN_PHASE_ONE, 
		typology						:= MESSAGE_TYPOLOGY_ABNORMAL, 
		process							:= prc, 
		CONVERSION_this					:= level_stop_asm);	
	
	digital_input_init(
		object_name						:= CONCAT(prc_path, '_feeder_faulted_di'), 
		polarity_direct					:= TRUE, 
		process							:= prc, 
		CONVERSION_this					:= feeder_faulted_di);
	
	digital_check_and_message_init(
		object_name						:= CONCAT(prc_path, '_feeder_faulted_dchk'), 
		alarm_if_input_off				:= FALSE, 
		alarm_delay						:= LEVEL_ALARM_DELAY_MS, 
		enabled_at_powerup				:= TRUE, 
		individual_reset				:= FALSE, 
		machine_reaction				:= MACHINE_REACTION_NO_STOP, 
		typology						:= MESSAGE_TYPOLOGY_OBligation, 
		process							:= prc, 
		CONVERSION_this					:= feeder_faulted_dchk);

	digital_check_add_di(
		di								:= feeder_faulted_di, 
		CONVERSION_this					:= feeder_faulted_dchk);		
END_IF

IF objects_running()
THEN
	process_cycle(prc);
	
	digital_check_cycle(level_ok_dchk);
	digital_check_cycle(ready_dchk);
	digital_check_cycle(feeder_faulted_dchk);
	digital_actuator_cycle(standby_sact);		
END_IF
END_ACTION

ACTION _read_process_image:
;
END_ACTION

ACTION _read_var_input:
;
END_ACTION

ACTION _set_runtime_properties:
standby_command := standby_req;
END_ACTION

ACTION _write_output:
;
END_ACTION

END_PROGRAM

// ---- Application/CSP/Case/Glue/csp_case_glue.TcPOU
(*********************************** G.D S.p.A. - Technical Department ***********************************
============= PROGRAM INFO ============
FOLDER:             TBD
MACHINES INVOLVED:  TBD 

============= DESCRIPTION =============
csp machine declaration

============= REVISIONS ===============
Date		Version	 	Author      	Description             
----------	-------		------------  	--------------------------------------------
2020/02/19 	0000.00	 	G.Imbriaco		First object declatation and purge function.
										TODO: 	- one_product_shot_req from machine logic
												- wait drive board firmware update to use object parameter
												- shift register reject information in case of error

**********************************************************************************************************)
(*$R process_ref := prc; $*)
PROGRAM csp_case_glue
VAR
	
	prc:											process;
	prc_path:										STRING;

	gd_glue:										BOOL := FALSE;
	
	Test_glue_bool:									bool:=false;
	one_product_shot_req:							BOOL:=FALSE; 
	purge_req:										BOOL:=FALSE;(*$P $*)
	purge_run_req:									BOOL:=FALSE;(*$P $*)
	p_purge_frequency_hz:							INT := 20;(*$P $*)

	purge_running:									message;	
	
	purge_position:									BOOL:=FALSE;
	run_position:									BOOL:=TRUE;

	purge_conditions:								BOOL;
	purge_command:									BOOL;
	purge_in_progress:								BOOL;(*$M $*)
	debug_purge:									BOOL;
	purge_frequency:								INT;
	auto_purge_request:								BOOL;
	
	product_presence_from_shift_bool:				BOOL;
	force_product_presence:							BOOL;
	
	enable_conditions:								BOOL;
	run_conditions:									BOOL;
	debug:											BOOL;
	
	glue_check_phase_old:							REAL;
	
	fsm_status:										csp_case_glue_status_enum;(*$M $*)
	fsm_next_status:								csp_case_glue_status_enum;
	fsm_enable_condition:							BOOL:=FALSE;
	debug_state_machine:							BOOL:=FALSE;
	debug_state_machine_one_step:					BOOL:=FALSE;
	
	fsm_status_NEW:									csp_case_glue_status_enum;(*$M $*)
	fsm_next_status_NEW:							csp_case_glue_status_enum;

	hmi_purge_active_cbtn:							command_button;
	hmi_purge_active_dpr:							BOOL:=FALSE; 
	hmi_purge_active_hgos:							hmi_graphic_object_status;
	
	purge_active_motcond:							motorization_conditioner;
	
	hmi_os_glue_upper_gun1_cbtn:					command_button;
	hmi_os_glue_upper_gun2_cbtn:					command_button;
	hmi_os_glue_lower_gun1_cbtn:					command_button;
	hmi_os_glue_lower_gun2_cbtn:					command_button;
	
	hmi_os_glue_upper_gun1_hgos:					hmi_graphic_object_status;
	hmi_os_glue_upper_gun2_hgos:					hmi_graphic_object_status;
	hmi_os_glue_lower_gun1_hgos:					hmi_graphic_object_status;
	hmi_os_glue_lower_gun2_hgos:					hmi_graphic_object_status;
	
	hmi_ls_glue_upper_gun1_cbtn:					command_button;
	hmi_ls_glue_upper_gun2_cbtn:					command_button;
	hmi_ls_glue_lower_gun1_cbtn:					command_button;
	hmi_ls_glue_lower_gun2_cbtn:					command_button;
	
	hmi_ls_glue_upper_gun1_hgos:					hmi_graphic_object_status;
	hmi_ls_glue_upper_gun2_hgos:					hmi_graphic_object_status;
	hmi_ls_glue_lower_gun1_hgos:					hmi_graphic_object_status;
	hmi_ls_glue_lower_gun2_hgos:					hmi_graphic_object_status;
	Test_purge_logic: 								BOOL := FALSE;
	
	case_at_glue_sr: 								INT := 27;
	toggle_eye: 									BOOL := FALSE;
	glue_pe_active:									BOOL;
	toggle_shift_reg: 								BOOL;
	glue_shift_active: 								BOOL := FALSE;
	
	glue_vm_phgen: 									phase_generator;
	
	glue_leading_upper_on: 							LREAL := 172;
	glue_leading_upper_off: 						LREAL := 202;
	glue_leading_upper_phwin: 						phase_window;
	
	glue_trailing_upper_on: 						LREAL := 294;
	glue_trailing_upper_off: 						LREAL := 340;
	glue_trailing_upper_phwin: 						phase_window;
	
	glue_head_offset:								LREAL := 71;
	
	glue_on: 										LREAL;
	
	glue_leading_lower_on: 							LREAL;
	glue_leading_lower_off: 						LREAL;
	glue_leading_lower_phwin: 						phase_window;
	
	glue_trailing_lower_on: 						LREAL;
	glue_trailing_lower_off: 						LREAL;
	glue_trailing_lower_phwin: 						phase_window;
	
	CONVERSION_MM_TO_DEG:							LREAL := 0.5905511811023622; //609.6mm = 24"
	
	hot_glue_bypass: 								BOOL :=FALSE; (*$P $*)
	os_upper_bypass_req:							BOOL:=FALSE;(*$P $*)
	os_lower_bypass_req:							BOOL:=FALSE;(*$P $*)
	ls_upper_bypass_req:							BOOL:=FALSE;(*$P $*)
	ls_lower_bypass_req:							BOOL:=FALSE;(*$P $*)
	
	(* NEW GLUE LOGIC *)
	os_case_at_glue_latch: 							BOOL := FALSE;
	ls_case_at_glue_latch: 							BOOL := FALSE;
	
	glue_strip_length_mm:							LREAL := 10; (*$P $*) // length of glue strip
	glue_strip_length_deg:							LREAL;
	less_glue_strip_mm:								LREAL := -1; // -1 at 17.2 AND 4 at 5
	less_glue_strip_deg:							LREAL;
	
	max_comp_deg:									LREAL;
	
	max_glue_strip_deg:								LREAL;
	current_deg_per_ms:								LREAL := 1;
	max_glue_time_ms:								UDINT;
	
	number_of_dots:									DINT; (*$P $*)
	dot_1_enable:									BOOL;
	dot_2_enable:									BOOL;
	dot_3_enable:									BOOL;
	dot_4_enable:									BOOL;
	dot_5_enable:									BOOL;
	dot_6_enable:									BOOL;
	
	os_upper_gun_1_enable:							BOOL := TRUE;
	os_upper_gun_2_enable:							BOOL := TRUE;
	os_lower_gun_1_enable:							BOOL := TRUE;
	os_lower_gun_2_enable:							BOOL := TRUE;
	
	ls_upper_gun_1_enable:							BOOL := TRUE;
	ls_upper_gun_2_enable:							BOOL := TRUE;
	ls_lower_gun_1_enable:							BOOL := TRUE;
	ls_lower_gun_2_enable:							BOOL := TRUE;
	
	os_upper_gun_1_on_tmr:							timer;
	os_upper_gun_2_on_tmr:							timer;
	os_lower_gun_1_on_tmr:							timer;
	os_lower_gun_2_on_tmr:							timer;
	
	ls_upper_gun_1_on_tmr:							timer;
	ls_upper_gun_2_on_tmr:							timer;
	ls_lower_gun_1_on_tmr:							timer;
	ls_lower_gun_2_on_tmr:							timer;
	
	
	(* OS START MM'S *)
	os_leading_upper_start_mm:						LREAL := 290; (*$P $*) // offest to start on upper leading
	os_leading_upper_start_deg:						LREAL;
	os_leading_lower_start_mm:						LREAL := 206; (*$P $*) // offest to start on lower leading
	os_leading_lower_start_deg:						LREAL;
	
	os_trailing_upper_start_mm: 					LREAL := 497; (*$P $*) // offest to start on upper trailing
	os_trailing_upper_start_deg:					LREAL;
	os_trailing_lower_start_mm:						LREAL := 413; (*$P $*) // offest to start on lower trailing
	os_trailing_lower_start_deg:					LREAL;
	
	(* OS LEADING FLAP PHASE WINDOWS *)
	os_leading_upper_dot_1_phwin:					phase_window;
	os_leading_upper_dot_2_phwin:					phase_window;
	os_leading_upper_dot_3_phwin:					phase_window;
	os_leading_upper_dot_4_phwin:					phase_window;
	os_leading_upper_dot_5_phwin:					phase_window;
	os_leading_upper_dot_6_phwin:					phase_window;
	
	os_leading_lower_dot_1_phwin:					phase_window;
	os_leading_lower_dot_2_phwin:					phase_window;
	os_leading_lower_dot_3_phwin:					phase_window;
	os_leading_lower_dot_4_phwin:					phase_window;
	os_leading_lower_dot_5_phwin:					phase_window;
	os_leading_lower_dot_6_phwin:					phase_window;
	
	(* OS TRAILING FLAP PHASE WINDOWS *)
	os_trailing_upper_dot_1_phwin:					phase_window;
	os_trailing_upper_dot_2_phwin:					phase_window;
	os_trailing_upper_dot_3_phwin:					phase_window;
	os_trailing_upper_dot_4_phwin:					phase_window;
	os_trailing_upper_dot_5_phwin:					phase_window;
	os_trailing_upper_dot_6_phwin:					phase_window;
	
	os_trailing_lower_dot_1_phwin:					phase_window;
	os_trailing_lower_dot_2_phwin:					phase_window;
	os_trailing_lower_dot_3_phwin:					phase_window;
	os_trailing_lower_dot_4_phwin:					phase_window;
	os_trailing_lower_dot_5_phwin:					phase_window;
	os_trailing_lower_dot_6_phwin:					phase_window;
	
	(* OS PHASE WINDOW ON OFFS *)
	os_leading_upper_dot_1_on:						LREAL;
	os_leading_upper_dot_1_on_comp:					LREAL;
	os_leading_upper_dot_1_off:						LREAL;
	os_leading_upper_dot_1_off_comp:				LREAL;
	os_leading_upper_dot_2_on:						LREAL;
	os_leading_upper_dot_2_on_comp:					LREAL;
	os_leading_upper_dot_2_off:						LREAL;
	os_leading_upper_dot_2_off_comp:				LREAL;
	os_leading_upper_dot_3_on:						LREAL;
	os_leading_upper_dot_3_on_comp:					LREAL;
	os_leading_upper_dot_3_off:						LREAL;
	os_leading_upper_dot_3_off_comp:				LREAL;
	os_leading_upper_dot_4_on:						LREAL;
	os_leading_upper_dot_4_on_comp:					LREAL;
	os_leading_upper_dot_4_off:						LREAL;
	os_leading_upper_dot_4_off_comp:				LREAL;
	os_leading_upper_dot_5_on:						LREAL;
	os_leading_upper_dot_5_on_comp:					LREAL;
	os_leading_upper_dot_5_off:						LREAL;
	os_leading_upper_dot_5_off_comp:				LREAL;
	os_leading_upper_dot_6_on:						LREAL;
	os_leading_upper_dot_6_on_comp:					LREAL;
	os_leading_upper_dot_6_off:						LREAL;
	os_leading_upper_dot_6_off_comp:				LREAL;
	
	os_leading_lower_dot_1_on:						LREAL;
	os_leading_lower_dot_1_on_comp:					LREAL;
	os_leading_lower_dot_1_off:						LREAL;
	os_leading_lower_dot_1_off_comp:				LREAL;
	os_leading_lower_dot_2_on:						LREAL;
	os_leading_lower_dot_2_on_comp:					LREAL;
	os_leading_lower_dot_2_off:						LREAL;
	os_leading_lower_dot_2_off_comp:				LREAL;
	os_leading_lower_dot_3_on:						LREAL;
	os_leading_lower_dot_3_on_comp:					LREAL;
	os_leading_lower_dot_3_off:						LREAL;
	os_leading_lower_dot_3_off_comp:				LREAL;
	os_leading_lower_dot_4_on:						LREAL;
	os_leading_lower_dot_4_on_comp:					LREAL;
	os_leading_lower_dot_4_off:						LREAL;
	os_leading_lower_dot_4_off_comp:				LREAL;
	os_leading_lower_dot_5_on:						LREAL;
	os_leading_lower_dot_5_on_comp:					LREAL;
	os_leading_lower_dot_5_off:						LREAL;
	os_leading_lower_dot_5_off_comp:				LREAL;
	os_leading_lower_dot_6_on:						LREAL;
	os_leading_lower_dot_6_on_comp:					LREAL;
	os_leading_lower_dot_6_off:						LREAL;
	os_leading_lower_dot_6_off_comp:				LREAL;
	
	os_trailing_upper_dot_1_on:						LREAL;
	os_trailing_upper_dot_1_on_comp:				LREAL;
	os_trailing_upper_dot_1_off:					LREAL;
	os_trailing_upper_dot_1_off_comp:				LREAL;
	os_trailing_upper_dot_2_on:						LREAL;
	os_trailing_upper_dot_2_on_comp:				LREAL;
	os_trailing_upper_dot_2_off:					LREAL;
	os_trailing_upper_dot_2_off_comp:				LREAL;
	os_trailing_upper_dot_3_on:						LREAL;
	os_trailing_upper_dot_3_on_comp:				LREAL;
	os_trailing_upper_dot_3_off:					LREAL;
	os_trailing_upper_dot_3_off_comp:				LREAL;
	os_trailing_upper_dot_4_on:						LREAL;
	os_trailing_upper_dot_4_on_comp:				LREAL;
	os_trailing_upper_dot_4_off:					LREAL;
	os_trailing_upper_dot_4_off_comp:				LREAL;
	os_trailing_upper_dot_5_on:						LREAL;
	os_trailing_upper_dot_5_on_comp:				LREAL;
	os_trailing_upper_dot_5_off:					LREAL;
	os_trailing_upper_dot_5_off_comp:				LREAL;
	os_trailing_upper_dot_6_on:						LREAL;
	os_trailing_upper_dot_6_on_comp:				LREAL;
	os_trailing_upper_dot_6_off:					LREAL;
	os_trailing_upper_dot_6_off_comp:				LREAL;
	
	os_trailing_lower_dot_1_on:						LREAL;
	os_trailing_lower_dot_1_on_comp:				LREAL;
	os_trailing_lower_dot_1_off:					LREAL;
	os_trailing_lower_dot_1_off_comp:				LREAL;
	os_trailing_lower_dot_2_on:						LREAL;
	os_trailing_lower_dot_2_on_comp:				LREAL;
	os_trailing_lower_dot_2_off:					LREAL;
	os_trailing_lower_dot_2_off_comp:				LREAL;
	os_trailing_lower_dot_3_on:						LREAL;
	os_trailing_lower_dot_3_on_comp:				LREAL;
	os_trailing_lower_dot_3_off:					LREAL;
	os_trailing_lower_dot_3_off_comp:				LREAL;
	os_trailing_lower_dot_4_on:						LREAL;
	os_trailing_lower_dot_4_on_comp:				LREAL;
	os_trailing_lower_dot_4_off:					LREAL;
	os_trailing_lower_dot_4_off_comp:				LREAL;
	os_trailing_lower_dot_5_on:						LREAL;
	os_trailing_lower_dot_5_on_comp:				LREAL;
	os_trailing_lower_dot_5_off:					LREAL;
	os_trailing_lower_dot_5_off_comp:				LREAL;
	os_trailing_lower_dot_6_on:						LREAL;
	os_trailing_lower_dot_6_on_comp:				LREAL;
	os_trailing_lower_dot_6_off:					LREAL;
	os_trailing_lower_dot_6_off_comp:				LREAL;
	
	
	(* LS START MM'S *)
	ls_leading_upper_start_mm:						LREAL := 290; (*$P $*) // offest to start on upper leading
	ls_leading_upper_start_deg:						LREAL;
	ls_leading_lower_start_mm:						LREAL := 206; (*$P $*) // offest to start on lower leading
	ls_leading_lower_start_deg:						LREAL;
	
	ls_trailing_upper_start_mm: 					LREAL := 497; (*$P $*) // offest to start on upper trailing
	ls_trailing_upper_start_deg:					LREAL;
	ls_trailing_lower_start_mm:						LREAL := 413; (*$P $*) // offest to start on lower trailing
	ls_trailing_lower_start_deg:					LREAL;
	
	(* LS LEADING FLAP PHASE WINDOWS *)
	ls_leading_upper_dot_1_phwin:					phase_window;
	ls_leading_upper_dot_2_phwin:					phase_window;
	ls_leading_upper_dot_3_phwin:					phase_window;
	ls_leading_upper_dot_4_phwin:					phase_window;
	ls_leading_upper_dot_5_phwin:					phase_window;
	ls_leading_upper_dot_6_phwin:					phase_window;
	
	ls_leading_lower_dot_1_phwin:					phase_window;
	ls_leading_lower_dot_2_phwin:					phase_window;
	ls_leading_lower_dot_3_phwin:					phase_window;
	ls_leading_lower_dot_4_phwin:					phase_window;
	ls_leading_lower_dot_5_phwin:					phase_window;
	ls_leading_lower_dot_6_phwin:					phase_window;
	
	(* LS TRAILING FLAP PHASE WINDOWS *)
	ls_trailing_upper_dot_1_phwin:					phase_window;
	ls_trailing_upper_dot_2_phwin:					phase_window;
	ls_trailing_upper_dot_3_phwin:					phase_window;
	ls_trailing_upper_dot_4_phwin:					phase_window;
	ls_trailing_upper_dot_5_phwin:					phase_window;
	ls_trailing_upper_dot_6_phwin:					phase_window;
	
	ls_trailing_lower_dot_1_phwin:					phase_window;
	ls_trailing_lower_dot_2_phwin:					phase_window;
	ls_trailing_lower_dot_3_phwin:					phase_window;
	ls_trailing_lower_dot_4_phwin:					phase_window;
	ls_trailing_lower_dot_5_phwin:					phase_window;
	ls_trailing_lower_dot_6_phwin:					phase_window;
	
	(* LS PHASE WINDOW ON OFFS *)
	ls_leading_upper_dot_1_on:						LREAL;
	ls_leading_upper_dot_1_on_comp:					LREAL;
	ls_leading_upper_dot_1_off:						LREAL;
	ls_leading_upper_dot_1_off_comp:				LREAL;
	ls_leading_upper_dot_2_on:						LREAL;
	ls_leading_upper_dot_2_on_comp:					LREAL;
	ls_leading_upper_dot_2_off:						LREAL;
	ls_leading_upper_dot_2_off_comp:				LREAL;
	ls_leading_upper_dot_3_on:						LREAL;
	ls_leading_upper_dot_3_on_comp:					LREAL;
	ls_leading_upper_dot_3_off:						LREAL;
	ls_leading_upper_dot_3_off_comp:				LREAL;
	ls_leading_upper_dot_4_on:						LREAL;
	ls_leading_upper_dot_4_on_comp:					LREAL;
	ls_leading_upper_dot_4_off:						LREAL;
	ls_leading_upper_dot_4_off_comp:				LREAL;
	ls_leading_upper_dot_5_on:						LREAL;
	ls_leading_upper_dot_5_on_comp:					LREAL;
	ls_leading_upper_dot_5_off:						LREAL;
	ls_leading_upper_dot_5_off_comp:				LREAL;
	ls_leading_upper_dot_6_on:						LREAL;
	ls_leading_upper_dot_6_on_comp:					LREAL;
	ls_leading_upper_dot_6_off:						LREAL;
	ls_leading_upper_dot_6_off_comp:				LREAL;
	
	ls_leading_lower_dot_1_on:						LREAL;
	ls_leading_lower_dot_1_on_comp:					LREAL;
	ls_leading_lower_dot_1_off:						LREAL;
	ls_leading_lower_dot_1_off_comp:				LREAL;
	ls_leading_lower_dot_2_on:						LREAL;
	ls_leading_lower_dot_2_on_comp:					LREAL;
	ls_leading_lower_dot_2_off:						LREAL;
	ls_leading_lower_dot_2_off_comp:				LREAL;
	ls_leading_lower_dot_3_on:						LREAL;
	ls_leading_lower_dot_3_on_comp:					LREAL;
	ls_leading_lower_dot_3_off:						LREAL;
	ls_leading_lower_dot_3_off_comp:				LREAL;
	ls_leading_lower_dot_4_on:						LREAL;
	ls_leading_lower_dot_4_on_comp:					LREAL;
	ls_leading_lower_dot_4_off:						LREAL;
	ls_leading_lower_dot_4_off_comp:				LREAL;
	ls_leading_lower_dot_5_on:						LREAL;
	ls_leading_lower_dot_5_on_comp:					LREAL;
	ls_leading_lower_dot_5_off:						LREAL;
	ls_leading_lower_dot_5_off_comp:				LREAL;
	ls_leading_lower_dot_6_on:						LREAL;
	ls_leading_lower_dot_6_on_comp:					LREAL;
	ls_leading_lower_dot_6_off:						LREAL;
	ls_leading_lower_dot_6_off_comp:				LREAL;
	
	ls_trailing_upper_dot_1_on:						LREAL;
	ls_trailing_upper_dot_1_on_comp:				LREAL;
	ls_trailing_upper_dot_1_off:					LREAL;
	ls_trailing_upper_dot_1_off_comp:				LREAL;
	ls_trailing_upper_dot_2_on:						LREAL;
	ls_trailing_upper_dot_2_on_comp:				LREAL;
	ls_trailing_upper_dot_2_off:					LREAL;
	ls_trailing_upper_dot_2_off_comp:				LREAL;
	ls_trailing_upper_dot_3_on:						LREAL;
	ls_trailing_upper_dot_3_on_comp:				LREAL;
	ls_trailing_upper_dot_3_off:					LREAL;
	ls_trailing_upper_dot_3_off_comp:				LREAL;
	ls_trailing_upper_dot_4_on:						LREAL;
	ls_trailing_upper_dot_4_on_comp:				LREAL;
	ls_trailing_upper_dot_4_off:					LREAL;
	ls_trailing_upper_dot_4_off_comp:				LREAL;
	ls_trailing_upper_dot_5_on:						LREAL;
	ls_trailing_upper_dot_5_on_comp:				LREAL;
	ls_trailing_upper_dot_5_off:					LREAL;
	ls_trailing_upper_dot_5_off_comp:				LREAL;
	ls_trailing_upper_dot_6_on:						LREAL;
	ls_trailing_upper_dot_6_on_comp:				LREAL;
	ls_trailing_upper_dot_6_off:					LREAL;
	ls_trailing_upper_dot_6_off_comp:				LREAL;
	
	ls_trailing_lower_dot_1_on:						LREAL;
	ls_trailing_lower_dot_1_on_comp:				LREAL;
	ls_trailing_lower_dot_1_off:					LREAL;
	ls_trailing_lower_dot_1_off_comp:				LREAL;
	ls_trailing_lower_dot_2_on:						LREAL;
	ls_trailing_lower_dot_2_on_comp:				LREAL;
	ls_trailing_lower_dot_2_off:					LREAL;
	ls_trailing_lower_dot_2_off_comp:				LREAL;
	ls_trailing_lower_dot_3_on:						LREAL;
	ls_trailing_lower_dot_3_on_comp:				LREAL;
	ls_trailing_lower_dot_3_off:					LREAL;
	ls_trailing_lower_dot_3_off_comp:				LREAL;
	ls_trailing_lower_dot_4_on:						LREAL;
	ls_trailing_lower_dot_4_on_comp:				LREAL;
	ls_trailing_lower_dot_4_off:					LREAL;
	ls_trailing_lower_dot_4_off_comp:				LREAL;
	ls_trailing_lower_dot_5_on:						LREAL;
	ls_trailing_lower_dot_5_on_comp:				LREAL;
	ls_trailing_lower_dot_5_off:					LREAL;
	ls_trailing_lower_dot_5_off_comp:				LREAL;
	ls_trailing_lower_dot_6_on:						LREAL;
	ls_trailing_lower_dot_6_on_comp:				LREAL;
	ls_trailing_lower_dot_6_off:					LREAL;
	ls_trailing_lower_dot_6_off_comp:				LREAL;
	
	(* NEW GLUE OUTPUTS *)
	os_upper_gun_1_do:								digital_output;
	os_upper_gun_2_do:								digital_output;
	os_lower_gun_1_do:								digital_output;
	os_lower_gun_2_do:								digital_output;
	
	ls_upper_gun_1_do:								digital_output;
	ls_upper_gun_2_do:								digital_output;
	ls_lower_gun_1_do:								digital_output;
	ls_lower_gun_2_do:								digital_output;
	
	enable_conditions_off: 							BOOL := FALSE;
	hmi_glue_ready_hgos:							hmi_graphic_object_status;
	hmi_glue_not_ready_hgos: 						hmi_graphic_object_status;
	OS_lower_glue_gun_disabled_wem:					message;					//PRS 7/14/2021
	OS_upper_glue_gun_disabled_wem:					message;					//PRS 7/14/2021
	LS_lower_glue_gun_disabled_wem:					message;					//PRS 7/14/2021
	LS_upper_glue_gun_disabled_wem:					message;					//PRS 7/14/2021
	absent_test: 									BOOL;
END_VAR

_read_var_input();

_object_manager();

IF NOT objects_running()
THEN
	RETURN;	
END_IF

_read_process_image();

_mode_manager();

CASE process_get_mode(prc) of
	MODE_ABSENT,
	MODE_INACTIVE:
		RETURN;
	MODE_TEST:
		_handle_process_test();
END_CASE

_set_runtime_properties();
absent_test := FALSE;
(********************************* BODY *********************************)
(* USED TO CHANGE VISIBILITY ON MESSAGE FOR RFID *)
IF NOT enable_conditions
	THEN
	enable_conditions_off := TRUE;
	ELSE
	enable_conditions_off := FALSE; 
END_IF


	hmi_graphic_object_set_status(
        status  			:= SEL(enable_conditions, HMI_OBJECT_STATUS_INVISIBLE, HMI_OBJECT_STATUS_ON),
        CONVERSION_this     := hmi_glue_ready_hgos);
	
	hmi_graphic_object_set_status(
        status  			:= SEL(enable_conditions_off, HMI_OBJECT_STATUS_ON, HMI_OBJECT_STATUS_INVISIBLE),
        CONVERSION_this     := hmi_glue_not_ready_hgos);
		
IF NOT purge_req
THEN
	motorization_conditioner_start_done(purge_active_motcond);
END_IF


(* UPPER LEADING FLAP PHWIN - MANUAL SET*)
phase_window_set_phases_data(
	begin_phase:=  glue_leading_upper_on,
	end_phase:=  glue_leading_upper_off,
	begin_delay:= 0,
	end_delay:= 0,
	begin_max_compensation:= 0,
	end_max_compensation:= 0,
	CONVERSION_this:= glue_leading_upper_phwin);

(* UPPER TRAILING FLAP PHWIN - MANUAL SET*)	
phase_window_set_phases_data(
    begin_phase:=  glue_trailing_upper_on,
    end_phase:=  glue_trailing_upper_off,
    begin_delay:= 0,
    end_delay:= 0,
    begin_max_compensation:= 0,
    end_max_compensation:= 0,
    CONVERSION_this:= glue_trailing_upper_phwin);

	
(* AUTO SET PHWIN OF LOWER BY GUN OFFSET *)
glue_leading_lower_on := glue_leading_upper_on - (CONVERSION_MM_TO_DEG * glue_head_offset);
glue_leading_lower_off := glue_leading_upper_off - (CONVERSION_MM_TO_DEG * glue_head_offset);

glue_trailing_lower_on := glue_trailing_upper_on - (CONVERSION_MM_TO_DEG * glue_head_offset);
glue_trailing_lower_off := glue_trailing_upper_off - (CONVERSION_MM_TO_DEG * glue_head_offset);		

	
(* LOWER LEADING FLAP PHWIN *)
phase_window_set_phases_data(
	begin_phase:=  glue_leading_lower_on,
	end_phase:=  glue_leading_lower_off,
	begin_delay:= 0,
	end_delay:= 0,
	begin_max_compensation:= 0,
	end_max_compensation:= 0,
	CONVERSION_this:= glue_leading_lower_phwin);
	
(* LOWER TRAILING FLAP PHWIN *)
phase_window_set_phases_data(
    begin_phase:=  glue_trailing_lower_on,
    end_phase:=  glue_trailing_lower_off,
    begin_delay:= 0,
    end_delay:= 0,
    begin_max_compensation:= 0,
    end_max_compensation:= 0,
    CONVERSION_this:= glue_trailing_lower_phwin);

	
(************************************************************************)

(**************************** PROGRAM HANDLER ***************************)

(* LOGIC TO DETERMINE IF GD OR BECKHOFF GLUE BOARDS *) (* GD Boards Removed *)

(* NEW GLUE CYCLE *)
_dot_calculations();
_run_cycle_NEW();



(* OS UPPER GUN 1 TIMEOUT *)
IF NOT digital_output_is_active(os_upper_gun_1_do)
	THEN
		timer_restart(max_glue_time_ms, os_upper_gun_1_on_tmr);
END_IF

IF	timer_is_expired(os_upper_gun_1_on_tmr)
	THEN
		digital_output_reset(os_upper_gun_1_do);
END_IF

(* OS UPPER GUN 2 TIMEOUT *)
IF NOT digital_output_is_active(os_upper_gun_2_do)
	THEN
		timer_restart(max_glue_time_ms, os_upper_gun_2_on_tmr);
END_IF

IF	timer_is_expired(os_upper_gun_2_on_tmr)
	THEN
		digital_output_reset(os_upper_gun_2_do);
END_IF

(* OS lower GUN 1 TIMEOUT *)
IF NOT digital_output_is_active(os_lower_gun_1_do)
	THEN
		timer_restart(max_glue_time_ms, os_lower_gun_1_on_tmr);
END_IF

IF	timer_is_expired(os_lower_gun_1_on_tmr)
	THEN
		digital_output_reset(os_lower_gun_1_do);
END_IF

(* OS lower GUN 2 TIMEOUT *)
IF NOT digital_output_is_active(os_lower_gun_2_do)
	THEN
		timer_restart(max_glue_time_ms, os_lower_gun_2_on_tmr);
END_IF

IF	timer_is_expired(os_lower_gun_2_on_tmr)
	THEN
		digital_output_reset(os_lower_gun_2_do);
END_IF


(* ls UPPER GUN 1 TIMEOUT *)
IF NOT digital_output_is_active(ls_upper_gun_1_do)
	THEN
		timer_restart(max_glue_time_ms, ls_upper_gun_1_on_tmr);
END_IF

IF	timer_is_expired(ls_upper_gun_1_on_tmr)
	THEN
		digital_output_reset(ls_upper_gun_1_do);
END_IF

(* ls UPPER GUN 2 TIMEOUT *)
IF NOT digital_output_is_active(ls_upper_gun_2_do)
	THEN
		timer_restart(max_glue_time_ms, ls_upper_gun_2_on_tmr);
END_IF

IF	timer_is_expired(ls_upper_gun_2_on_tmr)
	THEN
		digital_output_reset(ls_upper_gun_2_do);
END_IF

(* ls lower GUN 1 TIMEOUT *)
IF NOT digital_output_is_active(ls_lower_gun_1_do)
	THEN
		timer_restart(max_glue_time_ms, ls_lower_gun_1_on_tmr);
END_IF

IF	timer_is_expired(ls_lower_gun_1_on_tmr)
	THEN
		digital_output_reset(ls_lower_gun_1_do);
END_IF

(* ls lower GUN 2 TIMEOUT *)
IF NOT digital_output_is_active(ls_lower_gun_2_do)
	THEN
		timer_restart(max_glue_time_ms, ls_lower_gun_2_on_tmr);
END_IF

IF	timer_is_expired(ls_lower_gun_2_on_tmr)
	THEN
		digital_output_reset(ls_lower_gun_2_do);
END_IF

//PRS 7/14/2021
IF os_lower_bypass_req THEN
	process_message_set(1,1,1,OS_lower_glue_gun_disabled_wem);
ELSE
	process_message_reset(OS_lower_glue_gun_disabled_wem);
END_IF
IF os_upper_bypass_req THEN
	process_message_set(1,1,1,OS_upper_glue_gun_disabled_wem);
ELSE
	process_message_reset(OS_upper_glue_gun_disabled_wem);
END_IF
IF ls_lower_bypass_req THEN
	process_message_set(1,1,1,LS_lower_glue_gun_disabled_wem);
ELSE
	process_message_reset(LS_lower_glue_gun_disabled_wem);
END_IF
IF ls_upper_bypass_req THEN
	process_message_set(1,1,1,LS_upper_glue_gun_disabled_wem);
ELSE
	process_message_reset(LS_upper_glue_gun_disabled_wem);
END_IF


(************************************************************************)

_handle_messages();

_write_output();

ACTION _dot_calculations:
(* PHASE WINDOW CALCULATIONS *)
//upper_to_lower_offset_deg := upper_to_lower_offset_mm * CONVERSION_MM_TO_DEG;
glue_strip_length_deg := glue_strip_length_mm * CONVERSION_MM_TO_DEG;


// USED TO DETERMINE SPEED COMP
// NEED LOGIC HERE FOR THIS
max_comp_deg := -2 * CONVERSION_MM_TO_DEG;

IF csp_main_motorization_manager.motm.actual_velocity_setpoint > 20
	THEN
		less_glue_strip_deg := max_comp_deg;
ELSE
	less_glue_strip_deg := (-0.4098 * csp_main_motorization_manager.motm.actual_velocity + 6.0492) * CONVERSION_MM_TO_DEG;
END_IF


max_glue_strip_deg := glue_strip_length_deg + (-2.1 * max_comp_deg); (* -2.1 is to use 2 of the max comps for start and end and the .1 is for an extra amount in case a full timer is done *)

current_deg_per_ms := ((csp_main_motorization_manager.motm.actual_velocity_setpoint * 360) / 60) / 1000; (* Set point velocity * 360 degrees a cycle then divided by 60 to get degree per second then 1000 for degrees per ms *)

max_glue_time_ms := LREAL_TO_UDINT(max_glue_strip_deg / MAX(0.0001, current_deg_per_ms));


(* NUMBER OF DOTS *)
IF number_of_dots >= 1
THEN
	dot_1_enable := TRUE;
ELSE
	dot_1_enable := FALSE;
END_IF

IF number_of_dots >= 2
THEN
	dot_2_enable := TRUE;
ELSE
	dot_2_enable := FALSE;
END_IF

IF number_of_dots >= 3
THEN
	dot_3_enable := TRUE;
ELSE
	dot_3_enable := FALSE;
END_IF

IF number_of_dots >= 4
THEN
	dot_4_enable := TRUE;
ELSE
	dot_4_enable := FALSE;
END_IF

IF number_of_dots >= 5
THEN
	dot_5_enable := TRUE;
ELSE
	dot_5_enable := FALSE;
END_IF

IF number_of_dots >= 6
THEN
	dot_6_enable := TRUE;
ELSE
	dot_6_enable := FALSE;
END_IF



(* OS LEADING UPPER DOTS *)
os_leading_upper_start_deg := os_leading_upper_start_mm * CONVERSION_MM_TO_DEG;

os_leading_upper_dot_1_on := os_leading_upper_start_deg;
os_leading_upper_dot_1_off := os_leading_upper_dot_1_on + glue_strip_length_deg;

os_leading_upper_dot_2_on := os_leading_upper_dot_1_off + glue_strip_length_deg;
os_leading_upper_dot_2_off := os_leading_upper_dot_2_on + glue_strip_length_deg;

os_leading_upper_dot_3_on := os_leading_upper_dot_2_off + glue_strip_length_deg;
os_leading_upper_dot_3_off := os_leading_upper_dot_3_on + glue_strip_length_deg;

os_leading_upper_dot_4_on := os_leading_upper_dot_3_off + glue_strip_length_deg;
os_leading_upper_dot_4_off := os_leading_upper_dot_4_on + glue_strip_length_deg;

os_leading_upper_dot_5_on := os_leading_upper_dot_4_off + glue_strip_length_deg;
os_leading_upper_dot_5_off := os_leading_upper_dot_5_on + glue_strip_length_deg;

os_leading_upper_dot_6_on := os_leading_upper_dot_5_off + glue_strip_length_deg;
os_leading_upper_dot_6_off := os_leading_upper_dot_6_on + glue_strip_length_deg;

(* OS LEADING LOWER DOTS *)
os_leading_lower_start_deg := os_leading_lower_start_mm * CONVERSION_MM_TO_DEG;

os_leading_lower_dot_1_on := os_leading_lower_start_deg;
os_leading_lower_dot_1_off := os_leading_lower_dot_1_on + glue_strip_length_deg;

os_leading_lower_dot_2_on := os_leading_lower_dot_1_off + glue_strip_length_deg;
os_leading_lower_dot_2_off := os_leading_lower_dot_2_on + glue_strip_length_deg;

os_leading_lower_dot_3_on := os_leading_lower_dot_2_off + glue_strip_length_deg;
os_leading_lower_dot_3_off := os_leading_lower_dot_3_on + glue_strip_length_deg;

os_leading_lower_dot_4_on := os_leading_lower_dot_3_off + glue_strip_length_deg;
os_leading_lower_dot_4_off := os_leading_lower_dot_4_on + glue_strip_length_deg;

os_leading_lower_dot_5_on := os_leading_lower_dot_4_off + glue_strip_length_deg;
os_leading_lower_dot_5_off := os_leading_lower_dot_5_on + glue_strip_length_deg;

os_leading_lower_dot_6_on := os_leading_lower_dot_5_off + glue_strip_length_deg;
os_leading_lower_dot_6_off := os_leading_lower_dot_6_on + glue_strip_length_deg;


(* OS UPPER LEADING DOT 1 PHASE WINDOW *)
os_leading_upper_dot_1_on_comp := os_leading_upper_dot_1_on + less_glue_strip_deg;
os_leading_upper_dot_1_off_comp := os_leading_upper_dot_1_off - less_glue_strip_deg;

phase_window_set_phases_data(
	begin_phase:=  os_leading_upper_dot_1_on_comp,
	end_phase:=  os_leading_upper_dot_1_off_comp,
	begin_delay:= 0,
	end_delay:= 0,
	begin_max_compensation:= 0,
	end_max_compensation:= 0,
	CONVERSION_this:= os_leading_upper_dot_1_phwin);

(* OS UPPER LEADING DOT 2 PHASE WINDOW *)
os_leading_upper_dot_2_on_comp := os_leading_upper_dot_2_on + less_glue_strip_deg;
os_leading_upper_dot_2_off_comp := os_leading_upper_dot_2_off - less_glue_strip_deg;

phase_window_set_phases_data(
	begin_phase:=  os_leading_upper_dot_2_on_comp,
	end_phase:=  os_leading_upper_dot_2_off_comp,
	begin_delay:= 0,
	end_delay:= 0,
	begin_max_compensation:= 0,
	end_max_compensation:= 0,
	CONVERSION_this:= os_leading_upper_dot_2_phwin);

(* OS UPPER LEADING DOT 3 PHASE WINDOW *)
os_leading_upper_dot_3_on_comp := os_leading_upper_dot_3_on + less_glue_strip_deg;
os_leading_upper_dot_3_off_comp := os_leading_upper_dot_3_off - less_glue_strip_deg;

phase_window_set_phases_data(
	begin_phase:=  os_leading_upper_dot_3_on_comp,
	end_phase:=  os_leading_upper_dot_3_off_comp,
	begin_delay:= 0,
	end_delay:= 0,
	begin_max_compensation:= 0,
	end_max_compensation:= 0,
	CONVERSION_this:= os_leading_upper_dot_3_phwin);
	
(* OS UPPER LEADING DOT 4 PHASE WINDOW *)
os_leading_upper_dot_4_on_comp := os_leading_upper_dot_4_on + less_glue_strip_deg;
os_leading_upper_dot_4_off_comp := os_leading_upper_dot_4_off - less_glue_strip_deg;

phase_window_set_phases_data(
	begin_phase:=  os_leading_upper_dot_4_on_comp,
	end_phase:=  os_leading_upper_dot_4_off_comp,
	begin_delay:= 0,
	end_delay:= 0,
	begin_max_compensation:= 0,
	end_max_compensation:= 0,
	CONVERSION_this:= os_leading_upper_dot_4_phwin);

(* OS UPPER LEADING DOT 5 PHASE WINDOW *)
os_leading_upper_dot_5_on_comp := os_leading_upper_dot_5_on + less_glue_strip_deg;
os_leading_upper_dot_5_off_comp := os_leading_upper_dot_5_off - less_glue_strip_deg;

phase_window_set_phases_data(
	begin_phase:=  os_leading_upper_dot_5_on_comp,
	end_phase:=  os_leading_upper_dot_5_off_comp,
	begin_delay:= 0,
	end_delay:= 0,
	begin_max_compensation:= 0,
	end_max_compensation:= 0,
	CONVERSION_this:= os_leading_upper_dot_5_phwin);
	
(* OS UPPER LEADING DOT 6 PHASE WINDOW *)
os_leading_upper_dot_6_on_comp := os_leading_upper_dot_6_on + less_glue_strip_deg;
os_leading_upper_dot_6_off_comp := os_leading_upper_dot_6_off - less_glue_strip_deg;

phase_window_set_phases_data(
	begin_phase:=  os_leading_upper_dot_6_on_comp,
	end_phase:=  os_leading_upper_dot_6_off_comp,
	begin_delay:= 0,
	end_delay:= 0,
	begin_max_compensation:= 0,
	end_max_compensation:= 0,
	CONVERSION_this:= os_leading_upper_dot_6_phwin);
	
(* OS lower leading DOT 1 PHASE WINDOW *)
os_leading_lower_dot_1_on_comp := os_leading_lower_dot_1_on + less_glue_strip_deg;
os_leading_lower_dot_1_off_comp := os_leading_lower_dot_1_off - less_glue_strip_deg;

phase_window_set_phases_data(
	begin_phase:=  os_leading_lower_dot_1_on_comp,
	end_phase:=  os_leading_lower_dot_1_off_comp,
	begin_delay:= 0,
	end_delay:= 0,
	begin_max_compensation:= 0,
	end_max_compensation:= 0,
	CONVERSION_this:= os_leading_lower_dot_1_phwin);

(* OS lower leading DOT 2 PHASE WINDOW *)
os_leading_lower_dot_2_on_comp := os_leading_lower_dot_2_on + less_glue_strip_deg;
os_leading_lower_dot_2_off_comp := os_leading_lower_dot_2_off - less_glue_strip_deg;

phase_window_set_phases_data(
	begin_phase:=  os_leading_lower_dot_2_on_comp,
	end_phase:=  os_leading_lower_dot_2_off_comp,
	begin_delay:= 0,
	end_delay:= 0,
	begin_max_compensation:= 0,
	end_max_compensation:= 0,
	CONVERSION_this:= os_leading_lower_dot_2_phwin);

(* OS lower leading DOT 3 PHASE WINDOW *)
os_leading_lower_dot_3_on_comp := os_leading_lower_dot_3_on + less_glue_strip_deg;
os_leading_lower_dot_3_off_comp := os_leading_lower_dot_3_off - less_glue_strip_deg;

phase_window_set_phases_data(
	begin_phase:=  os_leading_lower_dot_3_on_comp,
	end_phase:=  os_leading_lower_dot_3_off_comp,
	begin_delay:= 0,
	end_delay:= 0,
	begin_max_compensation:= 0,
	end_max_compensation:= 0,
	CONVERSION_this:= os_leading_lower_dot_3_phwin);
	
(* OS lower leading DOT 4 PHASE WINDOW *)
os_leading_lower_dot_4_on_comp := os_leading_lower_dot_4_on + less_glue_strip_deg;
os_leading_lower_dot_4_off_comp := os_leading_lower_dot_4_off - less_glue_strip_deg;

phase_window_set_phases_data(
	begin_phase:=  os_leading_lower_dot_4_on_comp,
	end_phase:=  os_leading_lower_dot_4_off_comp,
	begin_delay:= 0,
	end_delay:= 0,
	begin_max_compensation:= 0,
	end_max_compensation:= 0,
	CONVERSION_this:= os_leading_lower_dot_4_phwin);

(* OS lower leading DOT 5 PHASE WINDOW *)
os_leading_lower_dot_5_on_comp := os_leading_lower_dot_5_on + less_glue_strip_deg;
os_leading_lower_dot_5_off_comp := os_leading_lower_dot_5_off - less_glue_strip_deg;

phase_window_set_phases_data(
	begin_phase:=  os_leading_lower_dot_5_on_comp,
	end_phase:=  os_leading_lower_dot_5_off_comp,
	begin_delay:= 0,
	end_delay:= 0,
	begin_max_compensation:= 0,
	end_max_compensation:= 0,
	CONVERSION_this:= os_leading_lower_dot_5_phwin);
	
(* OS lower leading DOT 6 PHASE WINDOW *)
os_leading_lower_dot_6_on_comp := os_leading_lower_dot_6_on + less_glue_strip_deg;
os_leading_lower_dot_6_off_comp := os_leading_lower_dot_6_off - less_glue_strip_deg;

phase_window_set_phases_data(
	begin_phase:=  os_leading_lower_dot_6_on_comp,
	end_phase:=  os_leading_lower_dot_6_off_comp,
	begin_delay:= 0,
	end_delay:= 0,
	begin_max_compensation:= 0,
	end_max_compensation:= 0,
	CONVERSION_this:= os_leading_lower_dot_6_phwin);
	
	
(* OS trailing UPPER DOTS *)
os_trailing_upper_start_deg := os_trailing_upper_start_mm * CONVERSION_MM_TO_DEG;

os_trailing_upper_dot_1_on := os_trailing_upper_start_deg;
os_trailing_upper_dot_1_off := os_trailing_upper_dot_1_on + glue_strip_length_deg;

os_trailing_upper_dot_2_on := os_trailing_upper_dot_1_off + glue_strip_length_deg;
os_trailing_upper_dot_2_off := os_trailing_upper_dot_2_on + glue_strip_length_deg;

os_trailing_upper_dot_3_on := os_trailing_upper_dot_2_off + glue_strip_length_deg;
os_trailing_upper_dot_3_off := os_trailing_upper_dot_3_on + glue_strip_length_deg;

os_trailing_upper_dot_4_on := os_trailing_upper_dot_3_off + glue_strip_length_deg;
os_trailing_upper_dot_4_off := os_trailing_upper_dot_4_on + glue_strip_length_deg;

os_trailing_upper_dot_5_on := os_trailing_upper_dot_4_off + glue_strip_length_deg;
os_trailing_upper_dot_5_off := os_trailing_upper_dot_5_on + glue_strip_length_deg;

os_trailing_upper_dot_6_on := os_trailing_upper_dot_5_off + glue_strip_length_deg;
os_trailing_upper_dot_6_off := os_trailing_upper_dot_6_on + glue_strip_length_deg;

(* OS trailing LOWER DOTS *)
os_trailing_lower_start_deg := os_trailing_lower_start_mm * CONVERSION_MM_TO_DEG;

os_trailing_lower_dot_1_on := os_trailing_lower_start_deg;
os_trailing_lower_dot_1_off := os_trailing_lower_dot_1_on + glue_strip_length_deg;

os_trailing_lower_dot_2_on := os_trailing_lower_dot_1_off + glue_strip_length_deg;
os_trailing_lower_dot_2_off := os_trailing_lower_dot_2_on + glue_strip_length_deg;

os_trailing_lower_dot_3_on := os_trailing_lower_dot_2_off + glue_strip_length_deg;
os_trailing_lower_dot_3_off := os_trailing_lower_dot_3_on + glue_strip_length_deg;

os_trailing_lower_dot_4_on := os_trailing_lower_dot_3_off + glue_strip_length_deg;
os_trailing_lower_dot_4_off := os_trailing_lower_dot_4_on + glue_strip_length_deg;

os_trailing_lower_dot_5_on := os_trailing_lower_dot_4_off + glue_strip_length_deg;
os_trailing_lower_dot_5_off := os_trailing_lower_dot_5_on + glue_strip_length_deg;

os_trailing_lower_dot_6_on := os_trailing_lower_dot_5_off + glue_strip_length_deg;
os_trailing_lower_dot_6_off := os_trailing_lower_dot_6_on + glue_strip_length_deg;

(* OS UPPER trailing DOT 1 PHASE WINDOW *)
os_trailing_upper_dot_1_on_comp := os_trailing_upper_dot_1_on + less_glue_strip_deg;
os_trailing_upper_dot_1_off_comp := os_trailing_upper_dot_1_off - less_glue_strip_deg;

phase_window_set_phases_data(
	begin_phase:=  os_trailing_upper_dot_1_on_comp,
	end_phase:=  os_trailing_upper_dot_1_off_comp,
	begin_delay:= 0,
	end_delay:= 0,
	begin_max_compensation:= 0,
	end_max_compensation:= 0,
	CONVERSION_this:= os_trailing_upper_dot_1_phwin);

(* OS UPPER trailing DOT 2 PHASE WINDOW *)
os_trailing_upper_dot_2_on_comp := os_trailing_upper_dot_2_on + less_glue_strip_deg;
os_trailing_upper_dot_2_off_comp := os_trailing_upper_dot_2_off - less_glue_strip_deg;

phase_window_set_phases_data(
	begin_phase:=  os_trailing_upper_dot_2_on_comp,
	end_phase:=  os_trailing_upper_dot_2_off_comp,
	begin_delay:= 0,
	end_delay:= 0,
	begin_max_compensation:= 0,
	end_max_compensation:= 0,
	CONVERSION_this:= os_trailing_upper_dot_2_phwin);

(* OS UPPER trailing DOT 3 PHASE WINDOW *)
os_trailing_upper_dot_3_on_comp := os_trailing_upper_dot_3_on + less_glue_strip_deg;
os_trailing_upper_dot_3_off_comp := os_trailing_upper_dot_3_off - less_glue_strip_deg;

phase_window_set_phases_data(
	begin_phase:=  os_trailing_upper_dot_3_on_comp,
	end_phase:=  os_trailing_upper_dot_3_off_comp,
	begin_delay:= 0,
	end_delay:= 0,
	begin_max_compensation:= 0,
	end_max_compensation:= 0,
	CONVERSION_this:= os_trailing_upper_dot_3_phwin);
	
(* OS UPPER trailing DOT 4 PHASE WINDOW *)
os_trailing_upper_dot_4_on_comp := os_trailing_upper_dot_4_on + less_glue_strip_deg;
os_trailing_upper_dot_4_off_comp := os_trailing_upper_dot_4_off - less_glue_strip_deg;

phase_window_set_phases_data(
	begin_phase:=  os_trailing_upper_dot_4_on_comp,
	end_phase:=  os_trailing_upper_dot_4_off_comp,
	begin_delay:= 0,
	end_delay:= 0,
	begin_max_compensation:= 0,
	end_max_compensation:= 0,
	CONVERSION_this:= os_trailing_upper_dot_4_phwin);

(* OS UPPER trailing DOT 5 PHASE WINDOW *)
os_trailing_upper_dot_5_on_comp := os_trailing_upper_dot_5_on + less_glue_strip_deg;
os_trailing_upper_dot_5_off_comp := os_trailing_upper_dot_5_off - less_glue_strip_deg;

phase_window_set_phases_data(
	begin_phase:=  os_trailing_upper_dot_5_on_comp,
	end_phase:=  os_trailing_upper_dot_5_off_comp,
	begin_delay:= 0,
	end_delay:= 0,
	begin_max_compensation:= 0,
	end_max_compensation:= 0,
	CONVERSION_this:= os_trailing_upper_dot_5_phwin);
	
(* OS UPPER trailing DOT 6 PHASE WINDOW *)
os_trailing_upper_dot_6_on_comp := os_trailing_upper_dot_6_on + less_glue_strip_deg;
os_trailing_upper_dot_6_off_comp := os_trailing_upper_dot_6_off - less_glue_strip_deg;

phase_window_set_phases_data(
	begin_phase:=  os_trailing_upper_dot_6_on_comp,
	end_phase:=  os_trailing_upper_dot_6_off_comp,
	begin_delay:= 0,
	end_delay:= 0,
	begin_max_compensation:= 0,
	end_max_compensation:= 0,
	CONVERSION_this:= os_trailing_upper_dot_6_phwin);
	
(* OS UPPER TRAILING DOT 1 PHASE WINDOW *)
os_trailing_lower_dot_1_on_comp := os_trailing_lower_dot_1_on + less_glue_strip_deg;
os_trailing_lower_dot_1_off_comp := os_trailing_lower_dot_1_off - less_glue_strip_deg;

phase_window_set_phases_data(
	begin_phase:=  os_trailing_lower_dot_1_on_comp,
	end_phase:=  os_trailing_lower_dot_1_off_comp,
	begin_delay:= 0,
	end_delay:= 0,
	begin_max_compensation:= 0,
	end_max_compensation:= 0,
	CONVERSION_this:= os_trailing_lower_dot_1_phwin);

(* OS UPPER TRAILING DOT 2 PHASE WINDOW *)
os_trailing_lower_dot_2_on_comp := os_trailing_lower_dot_2_on + less_glue_strip_deg;
os_trailing_lower_dot_2_off_comp := os_trailing_lower_dot_2_off - less_glue_strip_deg;

phase_window_set_phases_data(
	begin_phase:=  os_trailing_lower_dot_2_on_comp,
	end_phase:=  os_trailing_lower_dot_2_off_comp,
	begin_delay:= 0,
	end_delay:= 0,
	begin_max_compensation:= 0,
	end_max_compensation:= 0,
	CONVERSION_this:= os_trailing_lower_dot_2_phwin);

(* OS UPPER TRAILING DOT 3 PHASE WINDOW *)
os_trailing_lower_dot_3_on_comp := os_trailing_lower_dot_3_on + less_glue_strip_deg;
os_trailing_lower_dot_3_off_comp := os_trailing_lower_dot_3_off - less_glue_strip_deg;

phase_window_set_phases_data(
	begin_phase:=  os_trailing_lower_dot_3_on_comp,
	end_phase:=  os_trailing_lower_dot_3_off_comp,
	begin_delay:= 0,
	end_delay:= 0,
	begin_max_compensation:= 0,
	end_max_compensation:= 0,
	CONVERSION_this:= os_trailing_lower_dot_3_phwin);
	
(* OS UPPER TRAILING DOT 4 PHASE WINDOW *)
os_trailing_lower_dot_4_on_comp := os_trailing_lower_dot_4_on + less_glue_strip_deg;
os_trailing_lower_dot_4_off_comp := os_trailing_lower_dot_4_off - less_glue_strip_deg;

phase_window_set_phases_data(
	begin_phase:=  os_trailing_lower_dot_4_on_comp,
	end_phase:=  os_trailing_lower_dot_4_off_comp,
	begin_delay:= 0,
	end_delay:= 0,
	begin_max_compensation:= 0,
	end_max_compensation:= 0,
	CONVERSION_this:= os_trailing_lower_dot_4_phwin);

(* OS UPPER TRAILING DOT 5 PHASE WINDOW *)
os_trailing_lower_dot_5_on_comp := os_trailing_lower_dot_5_on + less_glue_strip_deg;
os_trailing_lower_dot_5_off_comp := os_trailing_lower_dot_5_off - less_glue_strip_deg;

phase_window_set_phases_data(
	begin_phase:=  os_trailing_lower_dot_5_on_comp,
	end_phase:=  os_trailing_lower_dot_5_off_comp,
	begin_delay:= 0,
	end_delay:= 0,
	begin_max_compensation:= 0,
	end_max_compensation:= 0,
	CONVERSION_this:= os_trailing_lower_dot_5_phwin);
	
(* OS UPPER TRAILING DOT 6 PHASE WINDOW *)
os_trailing_lower_dot_6_on_comp := os_trailing_lower_dot_6_on + less_glue_strip_deg;
os_trailing_lower_dot_6_off_comp := os_trailing_lower_dot_6_off - less_glue_strip_deg;

phase_window_set_phases_data(
	begin_phase:=  os_trailing_lower_dot_6_on_comp,
	end_phase:=  os_trailing_lower_dot_6_off_comp,
	begin_delay:= 0,
	end_delay:= 0,
	begin_max_compensation:= 0,
	end_max_compensation:= 0,
	CONVERSION_this:= os_trailing_lower_dot_6_phwin);
	
	
(* LS LEADING UPPER DOTS *)
ls_leading_upper_start_deg := ls_leading_upper_start_mm * CONVERSION_MM_TO_DEG;

ls_leading_upper_dot_1_on := ls_leading_upper_start_deg;
ls_leading_upper_dot_1_off := ls_leading_upper_dot_1_on + glue_strip_length_deg;

ls_leading_upper_dot_2_on := ls_leading_upper_dot_1_off + glue_strip_length_deg;
ls_leading_upper_dot_2_off := ls_leading_upper_dot_2_on + glue_strip_length_deg;

ls_leading_upper_dot_3_on := ls_leading_upper_dot_2_off + glue_strip_length_deg;
ls_leading_upper_dot_3_off := ls_leading_upper_dot_3_on + glue_strip_length_deg;

ls_leading_upper_dot_4_on := ls_leading_upper_dot_3_off + glue_strip_length_deg;
ls_leading_upper_dot_4_off := ls_leading_upper_dot_4_on + glue_strip_length_deg;

ls_leading_upper_dot_5_on := ls_leading_upper_dot_4_off + glue_strip_length_deg;
ls_leading_upper_dot_5_off := ls_leading_upper_dot_5_on + glue_strip_length_deg;

ls_leading_upper_dot_6_on := ls_leading_upper_dot_5_off + glue_strip_length_deg;
ls_leading_upper_dot_6_off := ls_leading_upper_dot_6_on + glue_strip_length_deg;

(* LS LEADING LOWER DOTS *)
ls_leading_lower_start_deg := ls_leading_lower_start_mm * CONVERSION_MM_TO_DEG;

ls_leading_lower_dot_1_on := ls_leading_lower_start_deg;
ls_leading_lower_dot_1_off := ls_leading_lower_dot_1_on + glue_strip_length_deg;

ls_leading_lower_dot_2_on := ls_leading_lower_dot_1_off + glue_strip_length_deg;
ls_leading_lower_dot_2_off := ls_leading_lower_dot_2_on + glue_strip_length_deg;

ls_leading_lower_dot_3_on := ls_leading_lower_dot_2_off + glue_strip_length_deg;
ls_leading_lower_dot_3_off := ls_leading_lower_dot_3_on + glue_strip_length_deg;

ls_leading_lower_dot_4_on := ls_leading_lower_dot_3_off + glue_strip_length_deg;
ls_leading_lower_dot_4_off := ls_leading_lower_dot_4_on + glue_strip_length_deg;

ls_leading_lower_dot_5_on := ls_leading_lower_dot_4_off + glue_strip_length_deg;
ls_leading_lower_dot_5_off := ls_leading_lower_dot_5_on + glue_strip_length_deg;

ls_leading_lower_dot_6_on := ls_leading_lower_dot_5_off + glue_strip_length_deg;
ls_leading_lower_dot_6_off := ls_leading_lower_dot_6_on + glue_strip_length_deg;


(* LS UPPER LEADING DOT 1 PHASE WINDOW *)
ls_leading_upper_dot_1_on_comp := ls_leading_upper_dot_1_on + less_glue_strip_deg;
ls_leading_upper_dot_1_off_comp := ls_leading_upper_dot_1_off - less_glue_strip_deg;

phase_window_set_phases_data(
	begin_phase:=  ls_leading_upper_dot_1_on_comp,
	end_phase:=  ls_leading_upper_dot_1_off_comp,
	begin_delay:= 0,
	end_delay:= 0,
	begin_max_compensation:= 0,
	end_max_compensation:= 0,
	CONVERSION_this:= ls_leading_upper_dot_1_phwin);

(* LS UPPER LEADING DOT 2 PHASE WINDOW *)
ls_leading_upper_dot_2_on_comp := ls_leading_upper_dot_2_on + less_glue_strip_deg;
ls_leading_upper_dot_2_off_comp := ls_leading_upper_dot_2_off - less_glue_strip_deg;

phase_window_set_phases_data(
	begin_phase:=  ls_leading_upper_dot_2_on_comp,
	end_phase:=  ls_leading_upper_dot_2_off_comp,
	begin_delay:= 0,
	end_delay:= 0,
	begin_max_compensation:= 0,
	end_max_compensation:= 0,
	CONVERSION_this:= ls_leading_upper_dot_2_phwin);

(* LS UPPER LEADING DOT 3 PHASE WINDOW *)
ls_leading_upper_dot_3_on_comp := ls_leading_upper_dot_3_on + less_glue_strip_deg;
ls_leading_upper_dot_3_off_comp := ls_leading_upper_dot_3_off - less_glue_strip_deg;

phase_window_set_phases_data(
	begin_phase:=  ls_leading_upper_dot_3_on_comp,
	end_phase:=  ls_leading_upper_dot_3_off_comp,
	begin_delay:= 0,
	end_delay:= 0,
	begin_max_compensation:= 0,
	end_max_compensation:= 0,
	CONVERSION_this:= ls_leading_upper_dot_3_phwin);
	
(* LS UPPER LEADING DOT 4 PHASE WINDOW *)
ls_leading_upper_dot_4_on_comp := ls_leading_upper_dot_4_on + less_glue_strip_deg;
ls_leading_upper_dot_4_off_comp := ls_leading_upper_dot_4_off - less_glue_strip_deg;

phase_window_set_phases_data(
	begin_phase:=  ls_leading_upper_dot_4_on_comp,
	end_phase:=  ls_leading_upper_dot_4_off_comp,
	begin_delay:= 0,
	end_delay:= 0,
	begin_max_compensation:= 0,
	end_max_compensation:= 0,
	CONVERSION_this:= ls_leading_upper_dot_4_phwin);

(* LS UPPER LEADING DOT 5 PHASE WINDOW *)
ls_leading_upper_dot_5_on_comp := ls_leading_upper_dot_5_on + less_glue_strip_deg;
ls_leading_upper_dot_5_off_comp := ls_leading_upper_dot_5_off - less_glue_strip_deg;

phase_window_set_phases_data(
	begin_phase:=  ls_leading_upper_dot_5_on_comp,
	end_phase:=  ls_leading_upper_dot_5_off_comp,
	begin_delay:= 0,
	end_delay:= 0,
	begin_max_compensation:= 0,
	end_max_compensation:= 0,
	CONVERSION_this:= ls_leading_upper_dot_5_phwin);
	
(* LS UPPER LEADING DOT 6 PHASE WINDOW *)
ls_leading_upper_dot_6_on_comp := ls_leading_upper_dot_6_on + less_glue_strip_deg;
ls_leading_upper_dot_6_off_comp := ls_leading_upper_dot_6_off - less_glue_strip_deg;

phase_window_set_phases_data(
	begin_phase:=  ls_leading_upper_dot_6_on_comp,
	end_phase:=  ls_leading_upper_dot_6_off_comp,
	begin_delay:= 0,
	end_delay:= 0,
	begin_max_compensation:= 0,
	end_max_compensation:= 0,
	CONVERSION_this:= ls_leading_upper_dot_6_phwin);
	
(* LS lower leading DOT 1 PHASE WINDOW *)
ls_leading_lower_dot_1_on_comp := ls_leading_lower_dot_1_on + less_glue_strip_deg;
ls_leading_lower_dot_1_off_comp := ls_leading_lower_dot_1_off - less_glue_strip_deg;

phase_window_set_phases_data(
	begin_phase:=  ls_leading_lower_dot_1_on_comp,
	end_phase:=  ls_leading_lower_dot_1_off_comp,
	begin_delay:= 0,
	end_delay:= 0,
	begin_max_compensation:= 0,
	end_max_compensation:= 0,
	CONVERSION_this:= ls_leading_lower_dot_1_phwin);

(* LS lower leading DOT 2 PHASE WINDOW *)
ls_leading_lower_dot_2_on_comp := ls_leading_lower_dot_2_on + less_glue_strip_deg;
ls_leading_lower_dot_2_off_comp := ls_leading_lower_dot_2_off - less_glue_strip_deg;

phase_window_set_phases_data(
	begin_phase:=  ls_leading_lower_dot_2_on_comp,
	end_phase:=  ls_leading_lower_dot_2_off_comp,
	begin_delay:= 0,
	end_delay:= 0,
	begin_max_compensation:= 0,
	end_max_compensation:= 0,
	CONVERSION_this:= ls_leading_lower_dot_2_phwin);

(* LS lower leading DOT 3 PHASE WINDOW *)
ls_leading_lower_dot_3_on_comp := ls_leading_lower_dot_3_on + less_glue_strip_deg;
ls_leading_lower_dot_3_off_comp := ls_leading_lower_dot_3_off - less_glue_strip_deg;

phase_window_set_phases_data(
	begin_phase:=  ls_leading_lower_dot_3_on_comp,
	end_phase:=  ls_leading_lower_dot_3_off_comp,
	begin_delay:= 0,
	end_delay:= 0,
	begin_max_compensation:= 0,
	end_max_compensation:= 0,
	CONVERSION_this:= ls_leading_lower_dot_3_phwin);
	
(* LS lower leading DOT 4 PHASE WINDOW *)
ls_leading_lower_dot_4_on_comp := ls_leading_lower_dot_4_on + less_glue_strip_deg;
ls_leading_lower_dot_4_off_comp := ls_leading_lower_dot_4_off - less_glue_strip_deg;

phase_window_set_phases_data(
	begin_phase:=  ls_leading_lower_dot_4_on_comp,
	end_phase:=  ls_leading_lower_dot_4_off_comp,
	begin_delay:= 0,
	end_delay:= 0,
	begin_max_compensation:= 0,
	end_max_compensation:= 0,
	CONVERSION_this:= ls_leading_lower_dot_4_phwin);

(* LS lower leading DOT 5 PHASE WINDOW *)
ls_leading_lower_dot_5_on_comp := ls_leading_lower_dot_5_on + less_glue_strip_deg;
ls_leading_lower_dot_5_off_comp := ls_leading_lower_dot_5_off - less_glue_strip_deg;

phase_window_set_phases_data(
	begin_phase:=  ls_leading_lower_dot_5_on_comp,
	end_phase:=  ls_leading_lower_dot_5_off_comp,
	begin_delay:= 0,
	end_delay:= 0,
	begin_max_compensation:= 0,
	end_max_compensation:= 0,
	CONVERSION_this:= ls_leading_lower_dot_5_phwin);
	
(* LS lower leading DOT 6 PHASE WINDOW *)
ls_leading_lower_dot_6_on_comp := ls_leading_lower_dot_6_on + less_glue_strip_deg;
ls_leading_lower_dot_6_off_comp := ls_leading_lower_dot_6_off - less_glue_strip_deg;

phase_window_set_phases_data(
	begin_phase:=  ls_leading_lower_dot_6_on_comp,
	end_phase:=  ls_leading_lower_dot_6_off_comp,
	begin_delay:= 0,
	end_delay:= 0,
	begin_max_compensation:= 0,
	end_max_compensation:= 0,
	CONVERSION_this:= ls_leading_lower_dot_6_phwin);
	
	
(* LS trailing UPPER DOTS *)
ls_trailing_upper_start_deg := ls_trailing_upper_start_mm * CONVERSION_MM_TO_DEG;

ls_trailing_upper_dot_1_on := ls_trailing_upper_start_deg;
ls_trailing_upper_dot_1_off := ls_trailing_upper_dot_1_on + glue_strip_length_deg;

ls_trailing_upper_dot_2_on := ls_trailing_upper_dot_1_off + glue_strip_length_deg;
ls_trailing_upper_dot_2_off := ls_trailing_upper_dot_2_on + glue_strip_length_deg;

ls_trailing_upper_dot_3_on := ls_trailing_upper_dot_2_off + glue_strip_length_deg;
ls_trailing_upper_dot_3_off := ls_trailing_upper_dot_3_on + glue_strip_length_deg;

ls_trailing_upper_dot_4_on := ls_trailing_upper_dot_3_off + glue_strip_length_deg;
ls_trailing_upper_dot_4_off := ls_trailing_upper_dot_4_on + glue_strip_length_deg;

ls_trailing_upper_dot_5_on := ls_trailing_upper_dot_4_off + glue_strip_length_deg;
ls_trailing_upper_dot_5_off := ls_trailing_upper_dot_5_on + glue_strip_length_deg;

ls_trailing_upper_dot_6_on := ls_trailing_upper_dot_5_off + glue_strip_length_deg;
ls_trailing_upper_dot_6_off := ls_trailing_upper_dot_6_on + glue_strip_length_deg;

(* LS trailing LOWER DOTS *)
ls_trailing_lower_start_deg := ls_trailing_lower_start_mm * CONVERSION_MM_TO_DEG;

ls_trailing_lower_dot_1_on := ls_trailing_lower_start_deg;
ls_trailing_lower_dot_1_off := ls_trailing_lower_dot_1_on + glue_strip_length_deg;

ls_trailing_lower_dot_2_on := ls_trailing_lower_dot_1_off + glue_strip_length_deg;
ls_trailing_lower_dot_2_off := ls_trailing_lower_dot_2_on + glue_strip_length_deg;

ls_trailing_lower_dot_3_on := ls_trailing_lower_dot_2_off + glue_strip_length_deg;
ls_trailing_lower_dot_3_off := ls_trailing_lower_dot_3_on + glue_strip_length_deg;

ls_trailing_lower_dot_4_on := ls_trailing_lower_dot_3_off + glue_strip_length_deg;
ls_trailing_lower_dot_4_off := ls_trailing_lower_dot_4_on + glue_strip_length_deg;

ls_trailing_lower_dot_5_on := ls_trailing_lower_dot_4_off + glue_strip_length_deg;
ls_trailing_lower_dot_5_off := ls_trailing_lower_dot_5_on + glue_strip_length_deg;

ls_trailing_lower_dot_6_on := ls_trailing_lower_dot_5_off + glue_strip_length_deg;
ls_trailing_lower_dot_6_off := ls_trailing_lower_dot_6_on + glue_strip_length_deg;

(* LS UPPER trailing DOT 1 PHASE WINDOW *)
ls_trailing_upper_dot_1_on_comp := ls_trailing_upper_dot_1_on + less_glue_strip_deg;
ls_trailing_upper_dot_1_off_comp := ls_trailing_upper_dot_1_off - less_glue_strip_deg;

phase_window_set_phases_data(
	begin_phase:=  ls_trailing_upper_dot_1_on_comp,
	end_phase:=  ls_trailing_upper_dot_1_off_comp,
	begin_delay:= 0,
	end_delay:= 0,
	begin_max_compensation:= 0,
	end_max_compensation:= 0,
	CONVERSION_this:= ls_trailing_upper_dot_1_phwin);

(* LS UPPER trailing DOT 2 PHASE WINDOW *)
ls_trailing_upper_dot_2_on_comp := ls_trailing_upper_dot_2_on + less_glue_strip_deg;
ls_trailing_upper_dot_2_off_comp := ls_trailing_upper_dot_2_off - less_glue_strip_deg;

phase_window_set_phases_data(
	begin_phase:=  ls_trailing_upper_dot_2_on_comp,
	end_phase:=  ls_trailing_upper_dot_2_off_comp,
	begin_delay:= 0,
	end_delay:= 0,
	begin_max_compensation:= 0,
	end_max_compensation:= 0,
	CONVERSION_this:= ls_trailing_upper_dot_2_phwin);

(* LS UPPER trailing DOT 3 PHASE WINDOW *)
ls_trailing_upper_dot_3_on_comp := ls_trailing_upper_dot_3_on + less_glue_strip_deg;
ls_trailing_upper_dot_3_off_comp := ls_trailing_upper_dot_3_off - less_glue_strip_deg;

phase_window_set_phases_data(
	begin_phase:=  ls_trailing_upper_dot_3_on_comp,
	end_phase:=  ls_trailing_upper_dot_3_off_comp,
	begin_delay:= 0,
	end_delay:= 0,
	begin_max_compensation:= 0,
	end_max_compensation:= 0,
	CONVERSION_this:= ls_trailing_upper_dot_3_phwin);
	
(* LS UPPER trailing DOT 4 PHASE WINDOW *)
ls_trailing_upper_dot_4_on_comp := ls_trailing_upper_dot_4_on + less_glue_strip_deg;
ls_trailing_upper_dot_4_off_comp := ls_trailing_upper_dot_4_off - less_glue_strip_deg;

phase_window_set_phases_data(
	begin_phase:=  ls_trailing_upper_dot_4_on_comp,
	end_phase:=  ls_trailing_upper_dot_4_off_comp,
	begin_delay:= 0,
	end_delay:= 0,
	begin_max_compensation:= 0,
	end_max_compensation:= 0,
	CONVERSION_this:= ls_trailing_upper_dot_4_phwin);

(* LS UPPER trailing DOT 5 PHASE WINDOW *)
ls_trailing_upper_dot_5_on_comp := ls_trailing_upper_dot_5_on + less_glue_strip_deg;
ls_trailing_upper_dot_5_off_comp := ls_trailing_upper_dot_5_off - less_glue_strip_deg;

phase_window_set_phases_data(
	begin_phase:=  ls_trailing_upper_dot_5_on_comp,
	end_phase:=  ls_trailing_upper_dot_5_off_comp,
	begin_delay:= 0,
	end_delay:= 0,
	begin_max_compensation:= 0,
	end_max_compensation:= 0,
	CONVERSION_this:= ls_trailing_upper_dot_5_phwin);
	
(* LS UPPER trailing DOT 6 PHASE WINDOW *)
ls_trailing_upper_dot_6_on_comp := ls_trailing_upper_dot_6_on + less_glue_strip_deg;
ls_trailing_upper_dot_6_off_comp := ls_trailing_upper_dot_6_off - less_glue_strip_deg;

phase_window_set_phases_data(
	begin_phase:=  ls_trailing_upper_dot_6_on_comp,
	end_phase:=  ls_trailing_upper_dot_6_off_comp,
	begin_delay:= 0,
	end_delay:= 0,
	begin_max_compensation:= 0,
	end_max_compensation:= 0,
	CONVERSION_this:= ls_trailing_upper_dot_6_phwin);
	
(* LS UPPER TRAILING DOT 1 PHASE WINDOW *)
ls_trailing_lower_dot_1_on_comp := ls_trailing_lower_dot_1_on + less_glue_strip_deg;
ls_trailing_lower_dot_1_off_comp := ls_trailing_lower_dot_1_off - less_glue_strip_deg;

phase_window_set_phases_data(
	begin_phase:=  ls_trailing_lower_dot_1_on_comp,
	end_phase:=  ls_trailing_lower_dot_1_off_comp,
	begin_delay:= 0,
	end_delay:= 0,
	begin_max_compensation:= 0,
	end_max_compensation:= 0,
	CONVERSION_this:= ls_trailing_lower_dot_1_phwin);

(* LS UPPER TRAILING DOT 2 PHASE WINDOW *)
ls_trailing_lower_dot_2_on_comp := ls_trailing_lower_dot_2_on + less_glue_strip_deg;
ls_trailing_lower_dot_2_off_comp := ls_trailing_lower_dot_2_off - less_glue_strip_deg;

phase_window_set_phases_data(
	begin_phase:=  ls_trailing_lower_dot_2_on_comp,
	end_phase:=  ls_trailing_lower_dot_2_off_comp,
	begin_delay:= 0,
	end_delay:= 0,
	begin_max_compensation:= 0,
	end_max_compensation:= 0,
	CONVERSION_this:= ls_trailing_lower_dot_2_phwin);

(* LS UPPER TRAILING DOT 3 PHASE WINDOW *)
ls_trailing_lower_dot_3_on_comp := ls_trailing_lower_dot_3_on + less_glue_strip_deg;
ls_trailing_lower_dot_3_off_comp := ls_trailing_lower_dot_3_off - less_glue_strip_deg;

phase_window_set_phases_data(
	begin_phase:=  ls_trailing_lower_dot_3_on_comp,
	end_phase:=  ls_trailing_lower_dot_3_off_comp,
	begin_delay:= 0,
	end_delay:= 0,
	begin_max_compensation:= 0,
	end_max_compensation:= 0,
	CONVERSION_this:= ls_trailing_lower_dot_3_phwin);
	
